// TwinCAT 3 PLC project CraneControl
// ProgramVersion: 3.1.4023.0
// libraries:
//   Tc2_Standard, * (Beckhoff Automation GmbH)
//   Tc2_System, * (Beckhoff Automation GmbH)
//   Tc3_Module, * (Beckhoff Automation GmbH)
//   VisuSymbols,3.5.10.0,System
// project tree:
//   ActuatorLimits/ FB_ActuatorLimits.TcPOU, FB_CartesianVelLimit.TcPOU, G_ActuatorLimits.TcGVL, P_ActuatorLimits.TcPOU, P_CartesianLimit.TcPOU
//   / Class Diagram.TcCD (not stored), GlobalTextList.TcGTLO, PlcTask.TcTTO, Visualization Manager.TcVMO (not stored)
//   ControlBox/ FB_AnalogInputScaling.TcPOU, FB_JoystickInputScaling.TcPOU, G_Buttons.TcGVL, G_ControlBoxInputs.TcGVL, G_Joystick.TcGVL, G_Outputs.TcGVL, G_ScalingParameters.TcGVL (not stored), P_JoystickInput.TcPOU, P_Outputs.TcPOU, ST_AnalogInput.TcDUT (not stored), ST_AnalogInputScaling.TcDUT (not stored), ST_AnalogInputStatus.TcDUT (not stored), ST_JoystickInputScaling.TcDUT (not stored), ST_Parameters.TcDUT
//   HeaveCompensation/ FB_Genr1b.TcPOU, FB_Get3r.TcPOU, G_Heave.TcGVL, P_Heave.TcPOU, P_SetZero.TcPOU
//   KinematicsForwAndInverseMatLab/ eps.TcPOU, eye.TcPOU, FB_ForwardKinematics.TcPOU, FB_InverseKinematics.TcPOU, isequal.TcPOU, MatrixLog3.TcPOU, norm.TcPOU, pinv.TcPOU, pinv_i.TcPOU, svd.TcPOU, svd_e.TcPOU, xaxpy.TcPOU, xaxpy_d.TcPOU, xaxpy_dm.TcPOU, xaxpy_dmy.TcPOU, xaxpy_dmyz.TcPOU, xaxpy_dmyzr.TcPOU, xaxpy_dmyzr5.TcPOU, xdotc.TcPOU, xdotc_i.TcPOU, xnrm2.TcPOU, xnrm2_l.TcPOU, xrot.TcPOU, xrotg.TcPOU, xrot_c.TcPOU, xrot_c5.TcPOU, xscal.TcPOU, xscal_f.TcPOU, xscal_fi.TcPOU, xscal_fiz.TcPOU, xscal_fiz1.TcPOU, rt_floord.TcPOU, rt_ldexp_U1d_U2s32_Yd_s_pw.TcPOU, xdotc_iq.TcPOU, xnrm2_l4.TcPOU, xnrm2_l4b.TcPOU, xscal_fiz1t.TcPOU, xscal_fiz1t4.TcPOU, xswap.TcPOU, xswap_g.TcPOU, xswap_gs.TcPOU
//   JoystickToCartesianVelocity/ FB_JoystickToCartesianVelocity.TcPOU
//   Kinematics_CraneFrame/ FB_ToolpointPositionIntegrator.TcPOU, G_InverseKinematics.TcGVL, G_Toolpoint.TcGVL, P_CartesianVelFromJoystick.TcPOU, P_Kinematics.TcPOU
//   PathGenerator/ FB_PathGenerator.TcPOU, G_Path.TcGVL, P_PathGeneration.TcPOU, P_PathGeneration_1.TcPOU, P_PathGeneration_2.TcPOU, P_PathGeneration_3.TcPOU
//   POUs/ MAIN.TcPOU, P_ModeControl.TcPOU, P_SlaveInputControl.TcPOU, Visualization.TcVIS
//   Sensors/ FB_DistSensorValue2Distance_q4.TcPOU, FB_Encoderval2Angle_q3.TcPOU, G_SensorInput.TcGVL, G_SensorsScaled.TcGVL, P_SensorScaling.TcPOU
//   ServoControl/ FB_PID.TcPOU, FB_PID_Controller.TcPOU, FB_ActuatorVelFeedForward.TcPOU, G_Servo.TcGVL, NormToPulseLenght.TcPOU, ButtonControlPulseLenght.TcPOU, P_CarteseanControllerServoActuation4DOF.TcPOU, P_ManualActuatorTest.TcPOU, P_NormalizeJointVel.TcPOU, P_CartesianController.TcPOU, P_Idle.TcPOU, P_ManualControl.TcPOU, P_VelToPos.TcPOU

CONFIGURATION CraneControl
    RESOURCE PLC ON TwinCAT3
        TASK PlcTask(INTERVAL := T#10ms, PRIORITY := 20);
        PROGRAM MAIN WITH PlcTask : MAIN;
    END_RESOURCE
END_CONFIGURATION

// ---- ControlBox/ST_Parameters.TcDUT
TYPE ST_Parameters :
STRUCT
	fCyclicTime 					: LREAL := 0.01; // [s]
	
	stJoystickInputScalingLeftX 		: ST_JoystickInputScaling := (fMaxInputValue := 20469.0, fMinInputValue := 11924.0, fNeutralInputValue := 16265, fNeutralDeadband := 100.0, fMaxOutputValue := 1.0, fMinOutputValue := -1.0, fNeutralOutputValue := 0.0);
	stJoystickInputScalingLeftY 		: ST_JoystickInputScaling := (fMaxInputValue := 20436.0, fMinInputValue := 11910.0, fNeutralInputValue := 16369, fNeutralDeadband := 100.0, fMaxOutputValue := 1.0, fMinOutputValue := -1.0, fNeutralOutputValue := 0.0);
	stJoystickInputScalingRightX 		: ST_JoystickInputScaling := (fMaxInputValue := 20481.0, fMinInputValue := 11905.0, fNeutralInputValue := 16370, fNeutralDeadband := 100.0, fMaxOutputValue := 1.0, fMinOutputValue := -1.0, fNeutralOutputValue := 0.0);
	stJoystickInputScalingRightY 		: ST_JoystickInputScaling := (fMaxInputValue := 20342.0, fMinInputValue := 12050.0, fNeutralInputValue := 16365, fNeutralDeadband := 100.0, fMaxOutputValue := 1.0, fMinOutputValue := -1.0, fNeutralOutputValue := 0.0);

		
END_STRUCT
END_TYPE

// ---- ActuatorLimits/G_ActuatorLimits.TcGVL
{attribute 'qualified_only'}
VAR_GLOBAL
	fq1Min: LREAL := -1.3;//rad
	fq1Max: LREAL := 1.3;//rad
	fq2Min: LREAL := -1.2;//rad 
	fq2Max: LREAL := 0.65;//rad
	fq3Min: LREAL := 0.15;//rad
	fq3Max: LREAL := 2.5;//rad
	fq4Min: LREAL := 0.0100;//m
	fq4Max: LREAL := 0.1900;//m

	bq1Min: BOOL;  // reached or not
	bq1Max: BOOL;
	bq2Min: BOOL;
	bq2Max: BOOL;
	bq3Min:	BOOL;
	bq3Max: BOOL;
	bq4Min: BOOL;
	bq4Max: BOOL;
	
	// Meassured in crane coordinates with tilt (theta = 0):
	fZMin : LREAL := -0.0500; //m 
	fZMax : LREAL := 0.4000;
	fYMin : LREAL := -0.25;
	fYMax : LREAL := 0.25;
	fXMax : LREAL := 0.45;
	fXMin : LREAL := 0.133;
END_VAR

// ---- ControlBox/G_Buttons.TcGVL
{attribute 'qualified_only'}
VAR_GLOBAL
	bManualModeSelector			AT %I* : BOOL;
	bAutoModeSelector			AT %I* : BOOL;
	//bRedButton					AT %I* : BOOL; Chaned fort extra button on joy stick
	//bGreenButton				AT %I* : BOOL; Chaned fort extra button on joy stick
	bJoystickLeftFrontEnable			AT %I* : BOOL;
	bJoystickRightFrontEnable			AT %I* : BOOL;
	bJoystickLeftEnable			AT %I* : BOOL;
	bJoystickRightEnable		AT %I* : BOOL;
	bSafetyRelayRestartButton   AT %I* : BOOL;
	
	// Analog Inputs
	stJoyLX 					: ST_AnalogInput;
	stJoyLY						: ST_AnalogInput;
	stJoyRX 					: ST_AnalogInput;
	stJoyRY						: ST_AnalogInput;

END_VAR

// ---- ControlBox/G_ControlBoxInputs.TcGVL
{attribute 'qualified_only'}
VAR_GLOBAL
	bManualModeSelector			AT %I* : BOOL;
	bAutoModeSelector			AT %I* : BOOL;
	bRedButton					AT %I* : BOOL;
	bGreenButton				AT %I* : BOOL;
	bJoystickLeftEnable			AT %I* : BOOL;
	bJoystickRightEnable		AT %I* : BOOL;
	bSafetyRelayRestartButton   AT %I* : BOOL;
	
	// Analog Inputs
	stJoyLX 					: ST_AnalogInput;
	stJoyLY						: ST_AnalogInput;
	stJoyRX 					: ST_AnalogInput;
	stJoyRY						: ST_AnalogInput;

END_VAR

// ---- ControlBox/G_Joystick.TcGVL
{attribute 'qualified_only'}
VAR_GLOBAL
	fJoystickLeftNormalizedY 		: LREAL;
	fJoystickLeftNormalizedX 		: LREAL;	
	fJoystickRightNormalizedY 		: LREAL;
	fJoystickRightNormalizedX 		: LREAL;
	
	nJoystickLeftDirectionX 		: DINT;
	nJoystickLeftDirectionY 		: DINT;
	nJoystickRightDirectionX 		: DINT;
	nJoystickRightDirectionY 		: DINT;
	
	bJoystick1InUse : BOOL ;
	bJoystick2InUse : BOOL;
	bJoystick3InUse : BOOL;
	bJoystick4InUse : BOOL;
		
END_VAR

// ---- ControlBox/G_Outputs.TcGVL
{attribute 'qualified_only'}
VAR_GLOBAL
	// PLC Rack
	
	// RIO Rack
	// Digital Outputs
	bGreenButtonLight 			AT %Q* : BOOL;
	bRedButtonLight 			AT %Q* : BOOL;
	// Analog Outputs
	//stWinchValveOutput 		: ST_ValveOutput;
	//stCylValveOutput 			: ST_ValveOutput;
	bSafetyRelayReset		 	AT %Q* : BOOL;
	
END_VAR

// ---- HeaveCompensation/G_Heave.TcGVL
{attribute 'qualified_only'}
VAR_GLOBAL
	fThetaStart : LREAL; //Tipping angle in degrees read at with system at rest
	fTheta : LREAL; //Tipping angle in degrees
	r3x : LREAL; //Vector from tipping point to toolpoint ref in frame coordinate
	r3y : LREAL; //Vector from tipping point to toolpoint ref in frame coordinate
	r3z : LREAL; //Vector from tipping point to toolpoint ref in frame coordinate
	r1bxCrane : LREAL; // Vector from crane base to toolpoint in Crane coordinates
	r1byCrane : LREAL; // Vector from crane base to toolpoint in Crane coordinates
	r1bzCrane : LREAL; // Vector from crane base to toolpoint in Crane coordinates
	bHeaveEnable : BOOL;
	bHeaveActive : BOOL := FALSE;
END_VAR

// ---- Kinematics_CraneFrame/G_InverseKinematics.TcGVL
{attribute 'qualified_only'}
VAR_GLOBAL
	fvXref  : LREAL; // Toolpoint cartesian velocity. From joistick. Used for inv. vel kin and calculate path for pos controller
	fvYref  : LREAL;
	fvZref  : LREAL;
	fq4Dotref : LREAL; //Actuator angular velocity from inverse vel kinematics m/s
	f_q1_ref : LREAL; //Ref angles from inverse position kinematics radians
	f_q2_ref : LREAL;
	f_q3_ref : LREAL;
	bKinematicsSucsessful : BOOL;
END_VAR

// ---- Kinematics_CraneFrame/G_Toolpoint.TcGVL
{attribute 'qualified_only'}
VAR_GLOBAL
	fX  : LREAL; //m
	fY  : LREAL; //m
	fZ  : LREAL; //m
	fXref  : LREAL; // Toolpoint cartesian reference signal position controller
	fYref  : LREAL;//m
	fZref  : LREAL;//m
END_VAR

// ---- PathGenerator/G_Path.TcGVL
{attribute 'qualified_only'}
VAR_GLOBAL
	bPathRunning  : BOOL;
	bPathFinnish : BOOL;
	bStartPath : BOOL;
	tTime : LREAL;
	bPathActivated : BOOL; // HMI path or Joistick
END_VAR

// ---- Sensors/G_SensorInput.TcGVL
{attribute 'qualified_only'}
VAR_GLOBAL
	fEncoder1Rad AT %I* : REAL;
	fEncoder2Rad AT %I* : REAL;
	fEncoder3Rad AT %I* : REAL;
	fTelescopeDistance_mm AT %I* : REAL;
	fXRotDeg AT %I* : REAL;
	fYRotDeg AT %I* : REAL;
	bSensorDataLost : BOOL;
END_VAR

// ---- Sensors/G_SensorsScaled.TcGVL
{attribute 'qualified_only'}
VAR_GLOBAL
	q1: REAL;
	q2  : REAL;
	q3  : REAL;
	q4 : REAL;
	q1Dot: REAL;
	q2Dot  : REAL;
	q3Dot  : REAL;
	q4Dot : REAL;
END_VAR

// ---- ServoControl/G_Servo.TcGVL
{attribute 'qualified_only'}
VAR_GLOBAL
	nServoPulseLenght1		AT %Q* : UINT;
	nServoPulseLenght2		AT %Q* : UINT;
	nServoPulseLenght3		AT %Q* : UINT;
	nServoPulseLenght4		AT %Q* : UINT;
	nServoPulseLenght5		AT %Q* : UINT;
	nServoPulseLenght6		AT %Q* : UINT;
	
	fNormalizedActuatorVelFeedForward_q1Dot : LREAL;
	fNormalizedActuatorVelFeedForward_q2Dot : LREAL;
	fNormalizedActuatorVelFeedForward_q3Dot : LREAL;
	fNormalizedActuatorVelFeedForward_q4Dot : LREAL;
	
	q1_position_error_part : LREAL;
	q2_position_error_part : LREAL;
	q3_position_error_part : LREAL;
	q4_position_error_part : LREAL;
	
	f_u_q1 :LREAL;
	f_u_q2 :LREAL;
	f_u_q3 :LREAL;
	f_u_q4 :LREAL; 
	
	
	//Temp for servo test:
	bStartSinus : BOOL;
	bSinusActive : BOOL;
	
END_VAR

// ---- POUs/MAIN.TcPOU
PROGRAM MAIN
VAR
END_VAR

P_ModeControl();

END_PROGRAM

// ---- POUs/P_ModeControl.TcPOU
PROGRAM P_ModeControl
VAR
	bAllowSinusInManualMode : BOOL;
END_VAR


// ONLY SET TRUE FOR ACTUATOR TEST IN MANUAL MODE:
bAllowSinusInManualMode := FALSE;



P_SensorScaling(); // Scaling sensor signals to mach q1,q2,q3,q4
P_Kinematics(); // Toolpoint position based on joint angles
P_JoystickInput(); // Normalize joistick signals from raw to -1 to 1


IF G_Buttons.bManualModeSelector AND NOT(G_Buttons.bAutoModeSelector) THEN // Manual mode
	
	//Only for actuationg the joints with open loop sinus
	IF G_Servo.bSinusActive AND bAllowSinusInManualMode THEN
		P_ManualActuatorTest();
	ELSE
		P_ManualControl();
	END_IF
	
	
	
	P_ActuatorLimits(); // Checking sensors and light lamps in HMI, preventing crashes is ONLY in auto mode
ELSIF NOT(G_Buttons.bManualModeSelector) AND G_Buttons.bAutoModeSelector AND NOT(G_SensorInput.bSensorDataLost) THEN // Auto Mode
	// Choose joystick OR PathGeneration

	IF G_Path.bPathActivated THEN
		//P_PathGeneration_1();  // 4 DOF
		P_PathGeneration_2();  // 4 DOF (3 dof test different telescope)
		//P_PathGeneration();  // 3 DOF
	ELSE
		P_CartesianVelFromJoystick();		
	END_IF

	
	P_CartesianLimit(); // Stops velocity ref if outside boundaries


	IF G_Heave.bHeaveEnable THEN
		P_Heave();
		G_Heave.bHeaveActive := TRUE;
	ELSE
		G_Heave.bHeaveActive := FALSE;
		P_VelToPos(); //Integrates pos to vel if 
	END_IF
	
	P_CartesianController();
ELSE // ModeButton in zero position
	P_Idle();
	P_SetZero();
	G_Heave.bHeaveActive := FALSE;
END_IF


P_Outputs(); //Lights on control box

END_PROGRAM

// ---- Sensors/P_SensorScaling.TcPOU
PROGRAM P_SensorScaling
VAR
		fbEncoderval2Angleq3 : FB_Encoderval2Angle_q3;
		fbDistSensorValue2Distance_q4 : FB_DistSensorValue2Distance_q4;

	
	// Temp variables for checking sensor comunication
	tempTOF1: LREAL;
	tempTOF11: LREAL;
	tempCounter: DINT := 0;

END_VAR

fbEncoderval2Angleq3(theta_i := G_SensorInput.fEncoder3Rad ,
					q3 => G_SensorsScaled.q3);
					
					
G_SensorsScaled.q1 := -G_SensorInput.fEncoder1Rad;
G_SensorsScaled.q2 := -G_SensorInput.fEncoder2Rad;



fbDistSensorValue2Distance_q4(fSensorValue := G_SensorInput.fTelescopeDistance_mm,
							f_q4 => G_SensorsScaled.q4);								
// TEMP FOR 3 DOF
//G_SensorsScaled.q4 := 0;
			

/////////////////////////////////////////////////////////////////////////////
// Check if sensors are comunicating and lighting RED LED communication lost	
tempTOF1 := G_SensorInput.fTelescopeDistance_mm;
IF tempTOF1 = tempTOF11 THEN
	tempCounter := tempCounter +1;
ELSE
	tempCounter := 0;
END_IF
tempTOF11 := G_SensorInput.fTelescopeDistance_mm;

IF tempCounter > 50 THEN
	G_SensorInput.bSensorDataLost := TRUE;
ELSE
	G_SensorInput.bSensorDataLost := FALSE;
END_IF
//////////////////////////////////////////////////////////////////////////////

END_PROGRAM

// ---- Sensors/FB_Encoderval2Angle_q3.TcPOU
FUNCTION_BLOCK FB_Encoderval2Angle_q3
VAR_INPUT
	theta_i: REAL;
END_VAR
VAR_OUTPUT
	q3: REAL;
END_VAR
VAR_TEMP
	ll: REAL;
	a: REAL;
	q3_tmp: REAL;
	temp1: REAL;
	temp2: REAL;
END_VAR

(* MATLAB Function: '<Root>/MATLAB Function' *)
(* Validated with physical measurements on crane from 0 - 180 deg *)
(* MATLAB Function 'MATLAB Function': '<S1>:1' *)
(* Constant Leght all mm: *)
(* '<S1>:1:6' theta_i_init = 2.3527; *)
(* start angle when piston is fully extracted *)
(* '<S1>:1:7' theta_k_init = 3.9706; *)
(* start angle when piston is fully extracted *)
(* '<S1>:1:8' Theta_I = theta_i_init + theta_i; *)
(* '<S1>:1:10' lh = 116.62; *)
(* '<S1>:1:11' li = 121.93; *)
(* '<S1>:1:12' lj = 13.34; *)
(* '<S1>:1:13' lk = 30; *)
(* '<S1>:1:14' lm = 20; *)
(* '<S1>:1:15' ln = 16; *)
(* '<S1>:1:16' theta_h = real(acos((lh^2+lj^2-li^2)/(2*lh*lj))); *)
(* Based on input: *)
(* Cylinder lenght: *)
(* '<S1>:1:20' xk = sqrt(lh^2+lk^2-2*lh*lk*cos(Theta_I)); *)

// PHMH ADDED BECAUSE BUNCTION DOES NOT HANDLE POSITIVE VALUES. Posistive values not possible after caluibration
IF theta_i >= 0 THEN
	theta_i := -0.00001;
ELSIF theta_i <= -1.5 THEN
	theta_i := -1.5;
END_IF




temp1 := COS(theta_i + 2.3527);
IF ABS(temp1) > 1 THEN
	temp1 := 1;
END_IF



a := SQRT(14500.224400000001 - (temp1 * 6997.2000000000007));
(* '<S1>:1:22' theta_j = theta_h-Theta_I; *)
(* '<S1>:1:23' ll = sqrt(lj^2+lk^2-2*lj*lk*cos(theta_j)); *)
temp2 := COS(1.9282807448254589 - (theta_i + 2.3527));
ll := SQRT(1077.9556 - (temp2 * 800.4));
(* '<S1>:1:25' theta_n = real(acos((ll^2+ln^2-lm^2)/(2*ll*ln))); *)
(* '<S1>:1:26' theta_l = acos((li^2+ll^2-xk^2)/(2*li*ll)); *)
(* '<S1>:1:27' theta_k = theta_n + theta_l; *)
(* '<S1>:1:28' q3 = theta_k-theta_k_init; *)
(* - init so output start at 0 *)
q3_tmp := ll * ll;
(* Outport: '<Root>/q3' incorporates:
 *  MATLAB Function: '<Root>/MATLAB Function' *)
q3 := -((ACOS(((q3_tmp + 256.0) - 400.0) / ((2.0 * ll) * 16.0)) + ACOS(((q3_tmp + 14866.924900000002) - (a * a)) / (243.86 * ll))) - 3.9706);

END_FUNCTION_BLOCK

// ---- Sensors/FB_DistSensorValue2Distance_q4.TcPOU
FUNCTION_BLOCK FB_DistSensorValue2Distance_q4
VAR_INPUT
	fSensorValue : REAL;
END_VAR
VAR_OUTPUT
	f_q4 : REAL;
END_VAR
VAR
DistSensorVal : REAL := 190; //mm
//Meassured value (Can be ecalibrated by looking in G_SensorInput and reading min and max telescope dist):
DistSensorMin : REAL  := 8.5; //mm
DistSensorMax : REAL := 193; //mm
 
q4Min : REAL := 167.25; //Maching with physical measurement 
q4Max : REAL := 367.25;//200 mm work space
END_VAR

f_q4 :=  ((fSensorValue-DistSensorMin)/(DistSensorMax-DistSensorMin)*(q4Max-q4Min))/1000;//m

END_FUNCTION_BLOCK

// ---- Kinematics_CraneFrame/P_Kinematics.TcPOU
PROGRAM P_Kinematics
VAR
fbForwardKinematics	: FB_ForwardKinematics;
END_VAR

fbForwardKinematics(q1 := G_SensorsScaled.q1, 
					q2 := G_SensorsScaled.q2,
					q3 := G_SensorsScaled.q3,
					q4 := G_SensorsScaled.q4,
					x => G_Toolpoint.fX,
					y => G_Toolpoint.fY,
					z => G_Toolpoint.fZ);

END_PROGRAM

// ---- KinematicsForwAndInverseMatLab/FB_ForwardKinematics.TcPOU
FUNCTION_BLOCK FB_ForwardKinematics
VAR_INPUT
    q1: LREAL;
    q2: LREAL;
    q3: LREAL;
    q4: LREAL;
END_VAR
VAR_OUTPUT
    x: LREAL;
    y: LREAL;
    z: LREAL;
END_VAR
VAR
    b: ARRAY [0..15] OF LREAL := [1.0,0.0,0.0,0.0,0.0,1.0,0.0,0.0,0.0,0.0,1.0,0.0,0.31920000000000004,0.02686,
        0.15515,1.0];
    c: ARRAY [0..35] OF LREAL := [0.0,0.0,1.0,0.0,0.0,0.0,0.0,1.0,0.0,-0.1569,0.0,-0.02745,0.0,1.0,0.0,-0.1569,0.0,
        0.15195,0.0,0.0,0.0,1.0,0.0,0.0,0.0,1.0,0.0,-0.15515,0.0,0.31920000000000004,0.0,0.0,1.0,0.02686,
        -0.31920000000000004,0.0];
    e_a: ARRAY [0..8] OF SINT := [1,0,0,0,1,0,0,0,1];
END_VAR
VAR_TEMP
    thetalist: ARRAY [0..5] OF LREAL;
    T: ARRAY [0..15] OF LREAL;
    i: DINT;
    se3mat: ARRAY [0..15] OF LREAL;
    omgmat: ARRAY [0..8] OF LREAL;
    a: ARRAY [0..15] OF LREAL;
    c_a: LREAL;
    V: ARRAY [0..5] OF LREAL;
    b_R: ARRAY [0..8] OF LREAL;
    b_omgmat: ARRAY [0..8] OF LREAL;
    d_a: LREAL;
    b_I: ARRAY [0..8] OF SINT;
    omgtheta_tmp: ARRAY [0..2] OF LREAL;
    thetalist_0: LREAL;
    a_0: ARRAY [0..15] OF LREAL;
    i_0: DINT;
    a_tmp_tmp: DINT;
    omgmat_tmp: DINT;
    R_tmp: DINT;
    c_a_tmp: LREAL;
    b_a_tmp: LREAL;
END_VAR

(* Lenght from assy drawing *)
(* MATLAB Function 'MATLAB Function': '<S1>:1' *)
(* '<S1>:1:4' l1 = 156.9/1000; *)
(* '<S1>:1:5' l2 = 27.45/1000; *)
(* '<S1>:1:6' l3 = 179.4/1000; *)
(* '<S1>:1:7' l4 = 26.86/1000; *)
(* From Telescope drawing (IN assy drawing) *)
(* l5 = 163.43;  *)
(* '<S1>:1:10' l5 = 167.25/1000; *)
(* Corrected after sensor calibration  *)
(* '<S1>:1:11' l6 = 1.75/1000; *)
(* mm *)
(* '<S1>:1:12' W1 = -l2+l3+l5; *)
(* '<S1>:1:13' W2 = l4; *)
(* '<S1>:1:14' W3 = l1-l6; *)
(* Position of each joint *)
(* '<S1>:1:18' a1 = [0; 0; 0]; *)
(* '<S1>:1:19' a2 = [-l2; 0; l1]; *)
(* '<S1>:1:20' a3 = [-l2+l3; 0; l1]; *)
(* '<S1>:1:21' a4 = [W1; W2; W3]; *)
(* '<S1>:1:22' a5 = [W1; W2; W3]; *)
(* '<S1>:1:23' a6 = [W1; W2; W3]; *)
(* Screw axis of ech joint *)
(* '<S1>:1:26' Sw1 = [0; 0; 1]; *)
(* '<S1>:1:27' Sw2 = [0; 1; 0]; *)
(* '<S1>:1:28' Sw3 = [0; 1; 0]; *)
(* '<S1>:1:29' Sw4 = [0; 0; 0]; *)
(* '<S1>:1:30' Sw5 = [0; 1; 0]; *)
(* '<S1>:1:31' Sw6 = [0; 0; 1]; *)
(* '<S1>:1:33' Sv1 = cross(a1,Sw1); *)
(* '<S1>:1:34' Sv2 = cross(a2,Sw2); *)
(* '<S1>:1:35' Sv3 = cross(a3,Sw3); *)
(* '<S1>:1:36' Sv4 = [1;0;0]; *)
(* translation along xaxis *)
(* '<S1>:1:37' Sv5 = cross(a5,Sw5); *)
(* '<S1>:1:38' Sv6 = cross(a6,Sw6); *)
(* '<S1>:1:40' S1 = [Sw1;Sv1]; *)
(* '<S1>:1:41' S2 = [Sw2;Sv2]; *)
(* '<S1>:1:42' S3 = [Sw3;Sv3]; *)
(* '<S1>:1:43' S4 = [Sw4;Sv4]; *)
(* '<S1>:1:44' S5 = [Sw5;Sv5]; *)
(* '<S1>:1:45' S6 = [Sw6;Sv6]; *)
(* '<S1>:1:47' M = [[1 0 0 W1]; *)
(* '<S1>:1:48'     [0 1 0 W2]; *)
(* '<S1>:1:49'     [0 0 1 W3]; *)
(* '<S1>:1:50'     [0 0 0 1];]; *)
(* MATLAB Function: '<Root>/MATLAB Function' *)
FOR i_0 := 0 TO 15 DO 
    T[i_0] := b[i_0];
END_FOR;
(* Joints:  *)
(* '<S1>:1:55' q5 = 0; *)
(* '<S1>:1:56' q6 = 0; *)
(* '<S1>:1:58' thetalist = [q1; q2 ; q3; q4; q5; q6]; *)
thetalist[0] := q1;
thetalist[1] := q2;
thetalist[2] := q3;
thetalist[3] := q4;
thetalist[4] := 0.0;
thetalist[5] := 0.0;
(* '<S1>:1:59' Slist = [S1,S2,S3,S4,S5,S6]; *)
(* '<S1>:1:63' T = M; *)
(* '<S1>:1:65' for i = 6: -1: 1 *)
(* MATLAB Function: '<Root>/MATLAB Function' *)
se3mat[0] := 0.0;
se3mat[5] := 0.0;
se3mat[10] := 0.0;
se3mat[3] := 0.0;
se3mat[7] := 0.0;
se3mat[11] := 0.0;
se3mat[15] := 0.0;
(* MATLAB Function: '<Root>/MATLAB Function' *)
(* MATLAB Function: '<Root>/MATLAB Function' *)
FOR i := 0 TO 5 DO 
    (* 6 = number of joints *)
    (* '<S1>:1:67' T = MatrixExp6(VecTose3(Slist(:, i) * thetalist(i))) * T; *)
    thetalist_0 := thetalist[5 - i];
    FOR i_0 := 0 TO 5 DO 
        V[i_0] := c[((5 - i) * 6) + i_0] * thetalist_0;
    END_FOR;
    (* *** CHAPTER 3: RIGID-BODY MOTIONS *** *)
    (* Takes a 6-vector (representing a spatial velocity). *)
    (* Returns the corresponding 4x4 se(3) matrix. *)
    (* Example Input: *)
    
    (* clear; clc; *)
    (* V = [1; 2; 3; 4; 5; 6]; *)
    (* se3mat = VecTose3(V) *)
    
    (* Output: *)
    (* se3mat = *)
    (* 0    -3     2     4 *)
    (* 3     0    -1     5 *)
    (* -2     1     0     6 *)
    (* 0     0     0     0  *)
    (* 'VecTose3:18' se3mat = [VecToso3(V(1: 3)), V(4: 6); 0, 0, 0, 0]; *)
    (* *** CHAPTER 3: RIGID-BODY MOTIONS *** *)
    (* Takes a 3-vector (angular velocity). *)
    (* Returns the skew symmetric matrix in so(3). *)
    (* Example Input: *)
    
    (* clear; clc; *)
    (* omg = [1; 2; 3]; *)
    (* so3mat = VecToso3(omg) *)
    
    (* Output: *)
    (* so3mat = *)
    (* 0    -3     2 *)
    (* 3     0    -1 *)
    (* -2     1     0 *)
    (* 'VecToso3:17' so3mat = [0, -omg(3), omg(2); omg(3), 0, -omg(1); -omg(2), omg(1), 0]; *)
    se3mat[4] :=  -V[2];
    se3mat[8] := V[1];
    se3mat[1] := V[2];
    se3mat[9] :=  -V[0];
    se3mat[2] :=  -V[1];
    se3mat[6] := V[0];
    se3mat[12] := V[3];
    se3mat[13] := V[4];
    se3mat[14] := V[5];
    (* *** CHAPTER 3: RIGID-BODY MOTIONS *** *)
    (* Takes a se(3) representation of exponential coordinates. *)
    (* Returns a T matrix in SE(3) that is achieved by traveling along/about the  *)
    (* screw axis S for a distance theta from an initial configuration T = I. *)
    (* Example Input: *)
    
    (* clear; clc; *)
    (* se3mat = [ 0,      0,       0,      0; *)
    (* 0,      0, -1.5708, 2.3562; *)
    (* 0, 1.5708,       0, 2.3562; *)
    (* 0,      0,       0,      0] *)
    (* T = MatrixExp6(se3mat) *)
    
    (* Output: *)
    (* T = *)
    (* 1.0000         0         0         0 *)
    (* 0    0.0000   -1.0000   -0.0000 *)
    (* 0    1.0000    0.0000    3.0000 *)
    (* 0         0         0    1.0000  *)
    (* 'MatrixExp6:22' omgtheta = so3ToVec(se3mat(1: 3, 1: 3)); *)
    (* *** CHAPTER 3: RIGID-BODY MOTIONS *** *)
    (* Takes a 3x3 skew-symmetric matrix (an element of so(3)). *)
    (* Returns the corresponding 3-vector (angular velocity). *)
    (* Example Input:  *)
    
    (* clear; clc; *)
    (* so3mat = [[0, -3, 2]; [3, 0, -1]; [-2, 1, 0]]; *)
    (* omg = so3ToVec(so3mat)   *)
    
    (* Output: *)
    (* omg = *)
    (* 1 *)
    (* 2 *)
    (* 3 *)
    (* 'so3ToVec:17' omg = [so3mat(3, 2); so3mat(1, 3); so3mat(2, 1)]; *)
    omgtheta_tmp[0] := V[0];
    omgtheta_tmp[1] := V[1];
    omgtheta_tmp[2] := V[2];
    (* 'MatrixExp6:23' if NearZero(norm(omgtheta)) *)
    (* *** BASIC HELPER FUNCTIONS *** *)
    (* Takes a scalar. *)
    (* Checks if the scalar is small enough to be neglected. *)
    (* Example Input: *)
    
    (* clear; clc; *)
    (* near = -1e-7; *)
    (* judge = NearZero(near) *)
    
    (* Output: *)
    (* judge = *)
    (* 1 *)
    (* 'NearZero:15' judge = norm(near) < 1e-6; *)
    thetalist_0 := norm(x := omgtheta_tmp);
    d_a := ABS(thetalist_0);
    IF d_a < 1.0E-6 THEN 
        (* 'MatrixExp6:24' T = [eye(3), se3mat(1: 3, 4); 0, 0, 0, 1]; *)
        FOR i_0 := 0 TO 8 DO 
            b_I[i_0] := 0;
        END_FOR;
        b_I[0] := 1;
        b_I[4] := 1;
        b_I[8] := 1;
        FOR i_0 := 0 TO 2 DO 
            R_tmp := DWORD_TO_DINT(SHL(DINT_TO_DWORD(i_0), 2));
            a[R_tmp] := SINT_TO_LREAL(b_I[3 * i_0]);
            a[R_tmp + 1] := SINT_TO_LREAL(b_I[(3 * i_0) + 1]);
            a[R_tmp + 2] := SINT_TO_LREAL(b_I[(3 * i_0) + 2]);
            a[i_0 + 12] := se3mat[i_0 + 12];
        END_FOR;
        a[3] := 0.0;
        a[7] := 0.0;
        a[11] := 0.0;
        a[15] := 1.0;
    ELSE 
        (* 'MatrixExp6:25' else *)
        (* 'MatrixExp6:26' [omghat, theta] = AxisAng3(omgtheta); *)
        (* *** CHAPTER 3: RIGID-BODY MOTIONS *** *)
        (* Takes A 3-vector of exponential coordinates for rotation. *)
        (* Returns the unit rotation axis omghat and the corresponding rotation  *)
        (* angle theta. *)
        (* Example Input: *)
        
        (* clear; clc; *)
        (* expc3 = [1; 2; 3]; *)
        (* [omghat, theta] = AxisAng3(expc3)   *)
        
        (* Output: *)
        (* omghat = *)
        (* 0.2673 *)
        (* 0.5345 *)
        (* 0.8018 *)
        (* theta = *)
        (* 3.7417 *)
        (* 'AxisAng3:20' theta = norm(expc3); *)
        (* 'AxisAng3:21' omghat = expc3 / theta; *)
        (* 'MatrixExp6:27' omgmat = se3mat(1: 3, 1: 3) / theta; *)
        FOR i_0 := 0 TO 2 DO 
            omgmat_tmp := DWORD_TO_DINT(SHL(DINT_TO_DWORD(i_0), 2));
            omgmat[3 * i_0] := se3mat[omgmat_tmp] / thetalist_0;
            omgmat[(3 * i_0) + 1] := se3mat[omgmat_tmp + 1] / thetalist_0;
            omgmat[(3 * i_0) + 2] := se3mat[omgmat_tmp + 2] / thetalist_0;
        END_FOR;
        (* 'MatrixExp6:28' T = [MatrixExp3(se3mat(1: 3, 1: 3)), ... *)
        (* 'MatrixExp6:29'          (eye(3) * theta + (1 - cos(theta)) * omgmat ... *)
        (* 'MatrixExp6:30'           + (theta - sin(theta)) * omgmat * omgmat) ... *)
        (* 'MatrixExp6:31'             * se3mat(1: 3, 4) / theta; *)
        (* 'MatrixExp6:32'          0, 0, 0, 1]; *)
        b_a_tmp := COS(thetalist_0);
        c_a_tmp := SIN(thetalist_0);
        c_a := thetalist_0 - c_a_tmp;
        (* *** CHAPTER 3: RIGID-BODY MOTIONS *** *)
        (* Takes a 3x3 so(3) representation of exponential coordinates. *)
        (* Returns R in SO(3) that is achieved by rotating about omghat by theta  *)
        (* from an initial orientation R = I. *)
        (* Example Input: *)
        
        (* clear; clc; *)
        (* so3mat = [[0, -3, 2]; [3, 0, -1]; [-2, 1, 0]]; *)
        (* R = MatrixExp3(so3mat)   *)
        
        (* Output: *)
        (* R = *)
        (* -0.6949    0.7135    0.0893 *)
        (* -0.1920   -0.3038    0.9332 *)
        (* 0.6930    0.6313    0.3481 *)
        (* 'MatrixExp3:18' omgtheta = so3ToVec(so3mat); *)
        (* *** CHAPTER 3: RIGID-BODY MOTIONS *** *)
        (* Takes a 3x3 skew-symmetric matrix (an element of so(3)). *)
        (* Returns the corresponding 3-vector (angular velocity). *)
        (* Example Input:  *)
        
        (* clear; clc; *)
        (* so3mat = [[0, -3, 2]; [3, 0, -1]; [-2, 1, 0]]; *)
        (* omg = so3ToVec(so3mat)   *)
        
        (* Output: *)
        (* omg = *)
        (* 1 *)
        (* 2 *)
        (* 3 *)
        (* 'so3ToVec:17' omg = [so3mat(3, 2); so3mat(1, 3); so3mat(2, 1)]; *)
        (* 'MatrixExp3:19' if NearZero(norm(omgtheta)) *)
        (* *** BASIC HELPER FUNCTIONS *** *)
        (* Takes a scalar. *)
        (* Checks if the scalar is small enough to be neglected. *)
        (* Example Input: *)
        
        (* clear; clc; *)
        (* near = -1e-7; *)
        (* judge = NearZero(near) *)
        
        (* Output: *)
        (* judge = *)
        (* 1 *)
        (* 'NearZero:15' judge = norm(near) < 1e-6; *)
        IF d_a < 1.0E-6 THEN 
            (* 'MatrixExp3:20' R = eye(3); *)
            FOR i_0 := 0 TO 8 DO 
                b_R[i_0] := 0.0;
            END_FOR;
            b_R[0] := 1.0;
            b_R[4] := 1.0;
            b_R[8] := 1.0;
        ELSE 
            (* 'MatrixExp3:21' else *)
            (* 'MatrixExp3:22' [omghat, theta] = AxisAng3(omgtheta); *)
            (* *** CHAPTER 3: RIGID-BODY MOTIONS *** *)
            (* Takes A 3-vector of exponential coordinates for rotation. *)
            (* Returns the unit rotation axis omghat and the corresponding rotation  *)
            (* angle theta. *)
            (* Example Input: *)
            
            (* clear; clc; *)
            (* expc3 = [1; 2; 3]; *)
            (* [omghat, theta] = AxisAng3(expc3)   *)
            
            (* Output: *)
            (* omghat = *)
            (* 0.2673 *)
            (* 0.5345 *)
            (* 0.8018 *)
            (* theta = *)
            (* 3.7417 *)
            (* 'AxisAng3:20' theta = norm(expc3); *)
            (* 'AxisAng3:21' omghat = expc3 / theta; *)
            (* 'MatrixExp3:23' omgmat = so3mat / theta; *)
            FOR i_0 := 0 TO 2 DO 
                omgmat_tmp := DWORD_TO_DINT(SHL(DINT_TO_DWORD(i_0), 2));
                b_omgmat[3 * i_0] := se3mat[omgmat_tmp] / thetalist_0;
                b_omgmat[(3 * i_0) + 1] := se3mat[omgmat_tmp + 1] / thetalist_0;
                b_omgmat[(3 * i_0) + 2] := se3mat[omgmat_tmp + 2] / thetalist_0;
            END_FOR;
            (* 'MatrixExp3:24' R = eye(3) + sin(theta) * omgmat + (1 - cos(theta)) * omgmat * omgmat; *)
            FOR i_0 := 0 TO 8 DO 
                b_I[i_0] := 0;
            END_FOR;
            b_I[0] := 1;
            b_I[4] := 1;
            b_I[8] := 1;
            FOR i_0 := 0 TO 2 DO 
                FOR omgmat_tmp := 0 TO 2 DO 
                    R_tmp := (3 * omgmat_tmp) + i_0;
                    b_R[R_tmp] := (((((1.0 - b_a_tmp) * b_omgmat[i_0 + 3]) * b_omgmat[(3 * omgmat_tmp) + 1]) + (((1.0 - b_a_tmp) * b_omgmat[i_0]) * b_omgmat[3 * omgmat_tmp])) + ((b_omgmat[i_0 + 6] * (1.0 - b_a_tmp)) * b_omgmat[(3 * omgmat_tmp) + 2])) + ((b_omgmat[R_tmp] * c_a_tmp) + SINT_TO_LREAL(b_I[R_tmp]));
                END_FOR;
            END_FOR;
        END_IF;
        FOR i_0 := 0 TO 2 DO 
            d_a := 0.0;
            FOR omgmat_tmp := 0 TO 2 DO 
                R_tmp := (3 * omgmat_tmp) + i_0;
                d_a := ((((((omgmat[i_0 + 3] * c_a) * omgmat[(3 * omgmat_tmp) + 1]) + ((c_a * omgmat[i_0]) * omgmat[3 * omgmat_tmp])) + ((omgmat[i_0 + 6] * c_a) * omgmat[(3 * omgmat_tmp) + 2])) + ((SINT_TO_LREAL(e_a[R_tmp]) * thetalist_0) + (omgmat[R_tmp] * (1.0 - b_a_tmp)))) * se3mat[omgmat_tmp + 12]) + d_a;
                a[omgmat_tmp + (i_0 * 4)] := b_R[(3 * i_0) + omgmat_tmp];
            END_FOR;
            a[i_0 + 12] := d_a / thetalist_0;
        END_FOR;
        a[3] := 0.0;
        a[7] := 0.0;
        a[11] := 0.0;
        a[15] := 1.0;
    END_IF;
    FOR i_0 := 0 TO 3 DO 
        FOR omgmat_tmp := 0 TO 3 DO 
            a_tmp_tmp := DWORD_TO_DINT(SHL(DINT_TO_DWORD(omgmat_tmp), 2));
            R_tmp := i_0 + a_tmp_tmp;
            a_0[R_tmp] := 0.0;
            a_0[R_tmp] := a_0[R_tmp] + (T[a_tmp_tmp] * a[i_0]);
            a_0[R_tmp] := (T[a_tmp_tmp + 1] * a[i_0 + 4]) + a_0[R_tmp];
            a_0[R_tmp] := (T[a_tmp_tmp + 2] * a[i_0 + 8]) + a_0[R_tmp];
            a_0[R_tmp] := (T[a_tmp_tmp + 3] * a[i_0 + 12]) + a_0[R_tmp];
        END_FOR;
    END_FOR;
    FOR i_0 := 0 TO 15 DO 
        T[i_0] := a_0[i_0];
    END_FOR;
END_FOR;
(* Outport: '<Root>/x' incorporates:
 *  MATLAB Function: '<Root>/MATLAB Function' *)
(* '<S1>:1:69' x = T(1,4); *)
(* '<S1>:1:70' y = T(2,4); *)
(* '<S1>:1:71' z = T(3,4); *)
x := T[12];
(* Outport: '<Root>/y' incorporates:
 *  MATLAB Function: '<Root>/MATLAB Function' *)
y := T[13];
(* Outport: '<Root>/z' incorporates:
 *  MATLAB Function: '<Root>/MATLAB Function' *)
z := T[14];

END_FUNCTION_BLOCK

// ---- KinematicsForwAndInverseMatLab/norm.TcPOU
FUNCTION norm : LREAL
VAR_INPUT
    x: ARRAY [0..2] OF LREAL;
END_VAR
VAR
    scale: LREAL;
    absxk: LREAL;
    t: LREAL;
END_VAR

scale := 3.3121686421112381E-170;
absxk := ABS(x[0]);
IF absxk > 3.3121686421112381E-170 THEN 
    norm := 1.0;
    scale := absxk;
ELSE 
    t := absxk / 3.3121686421112381E-170;
    norm := t * t;
END_IF;
absxk := ABS(x[1]);
IF absxk > scale THEN 
    t := scale / absxk;
    norm := ((norm * t) * t) + 1.0;
    scale := absxk;
ELSE 
    t := absxk / scale;
    norm := (t * t) + norm;
END_IF;
absxk := ABS(x[2]);
IF absxk > scale THEN 
    t := scale / absxk;
    norm := ((norm * t) * t) + 1.0;
    scale := absxk;
ELSE 
    t := absxk / scale;
    norm := (t * t) + norm;
END_IF;
norm := scale * SQRT(norm);

END_FUNCTION

// ---- ControlBox/P_JoystickInput.TcPOU
PROGRAM P_JoystickInput
VAR
	fbJoystickLeftVert 					: FB_JoystickInputScaling;
	fbJoystickLeftHor 					: FB_JoystickInputScaling;
	
	fbJoystickRightVert 				: FB_JoystickInputScaling;
	fbJoystickRightHor 					: FB_JoystickInputScaling;
	
	bEnableJoystick : BOOL;
		
END_VAR

bEnableJoystick := G_Buttons.bManualModeSelector OR G_Buttons.bAutoModeSelector;

fbJoystickLeftVert(
	bEnable := bEnableJoystick,
	nRawInput := G_Buttons.stJoyLY.nValue,
	stJoystickInputScaling := G_ScalingParameters.stParam.stJoystickInputScalingLeftY,
	fNormalizedOutput => G_Joystick.fJoystickLeftNormalizedY
);

IF G_Joystick.fJoystickLeftNormalizedY < 0 THEN
	G_Joystick.nJoystickLeftDirectionY := -1;
ELSIF G_Joystick.fJoystickLeftNormalizedY > 0 THEN
	G_Joystick.nJoystickLeftDirectionY := 1;	
END_IF

fbJoystickLeftHor(
	bEnable := bEnableJoystick,
	nRawInput := G_Buttons.stJoyLX.nValue,
	stJoystickInputScaling := G_ScalingParameters.stParam.stJoystickInputScalingLeftX,
	fNormalizedOutput => G_Joystick.fJoystickLeftNormalizedX
);

IF G_Joystick.fJoystickLeftNormalizedX < 0 THEN
	G_Joystick.nJoystickLeftDirectionX := 1;
ELSIF G_Joystick.fJoystickLeftNormalizedX > 0 THEN
	G_Joystick.nJoystickLeftDirectionX := -1;	
END_IF


fbJoystickRightVert(
	bEnable := bEnableJoystick,
	nRawInput := G_Buttons.stJoyRY.nValue,
	stJoystickInputScaling := G_ScalingParameters.stParam.stJoystickInputScalingRightY,
	fNormalizedOutput => G_Joystick.fJoystickRightNormalizedY
);

IF G_Joystick.fJoystickRightNormalizedY > 0 THEN
	G_Joystick.nJoystickRightDirectionY := -1;
ELSIF G_Joystick.fJoystickRightNormalizedY < 0 THEN
	G_Joystick.nJoystickRightDirectionY := 1;	
END_IF



fbJoystickRightHor(
	bEnable := bEnableJoystick,
	nRawInput := G_Buttons.stJoyRX.nValue,
	stJoystickInputScaling := G_ScalingParameters.stParam.stJoystickInputScalingRightX,
	fNormalizedOutput => G_Joystick.fJoystickRightNormalizedX
);

IF G_Joystick.fJoystickRightNormalizedX < 0 THEN
	G_Joystick.nJoystickRightDirectionX := 1;
ELSIF G_Joystick.fJoystickRightNormalizedX > 0 THEN
	G_Joystick.nJoystickRightDirectionX := -1;	
END_IF


// Activate bool for each joystick
IF G_Joystick.fJoystickRightNormalizedX < 0 OR G_Joystick.fJoystickRightNormalizedX > 0 THEN
	G_Joystick.bJoystick1InUse := TRUE;
ELSE
	G_Joystick.bJoystick1InUse := FALSE;
END_IF

IF G_Joystick.fJoystickRightNormalizedY < 0 OR G_Joystick.fJoystickRightNormalizedY > 0 THEN
	G_Joystick.bJoystick2InUse := TRUE;
ELSE
	G_Joystick.bJoystick2InUse := FALSE;
END_IF

IF G_Joystick.fJoystickLeftNormalizedX < 0 OR G_Joystick.fJoystickLeftNormalizedX > 0 THEN
	G_Joystick.bJoystick3InUse := TRUE;
ELSE
	G_Joystick.bJoystick3InUse := FALSE;
END_IF

IF G_Joystick.fJoystickLeftNormalizedY < 0 OR G_Joystick.fJoystickLeftNormalizedY > 0 THEN
	G_Joystick.bJoystick4InUse := TRUE;
ELSE
	G_Joystick.bJoystick4InUse := FALSE;
END_IF

END_PROGRAM

// ---- ControlBox/FB_JoystickInputScaling.TcPOU
FUNCTION_BLOCK FB_JoystickInputScaling
VAR_INPUT
	bEnable  : BOOL;
	nRawInput : INT;
	stJoystickInputScaling : ST_JoystickInputScaling;
END_VAR
VAR_OUTPUT
	fNormalizedOutput : LREAL;
END_VAR
VAR
	fRawInput : LREAL;
	fTempInput : LREAL;
	fTempOutput : LREAL;
END_VAR

fRawInput := INT_TO_REAL(nRawInput);

fTempInput := fRawInput - stJoystickInputScaling.fNeutralInputValue;
IF fTempInput > stJoystickInputScaling.fNeutralDeadband THEN
	fTempOutput := fTempInput/(stJoystickInputScaling.fMaxInputValue - stJoystickInputScaling.fNeutralInputValue);
ELSIF fTempInput < -stJoystickInputScaling.fNeutralDeadband THEN
	fTempOutput := fTempInput/(stJoystickInputScaling.fNeutralInputValue - stJoystickInputScaling.fMinInputValue);
ELSE
	fTempOutput := 0;
END_IF

IF nRawInput = 0 THEN
	fNormalizedOutput := -0.0;
ELSIF NOT (bEnable) THEN
	fNormalizedOutput := -0.0;
ELSE 
	fNormalizedOutput := LIMIT(stJoystickInputScaling.fMinOutputValue, fTempOutput, stJoystickInputScaling.fMaxOutputValue);
END_IF

END_FUNCTION_BLOCK

// ---- ServoControl/P_ManualActuatorTest.TcPOU
PROGRAM P_ManualActuatorTest
VAR
	fbPathGenerator: FB_PathGenerator;
	Q1: BOOL;
	t: INT;
	ElapsedTime : LREAL;
	sinus :  LREAL;
	nsinus : UINT;
END_VAR

// This program is used only to make results for the manual controller. 
//Actuating each joint with sinusoidal wave and check the sensor


fbPathGenerator(bStart := G_Servo.bStartSinus, 
				TIN := T#15S , 
				Qout =>Q1, 
				t => ElapsedTime);
sinus := 70*SIN(ElapsedTime*2/2);
nsinus :=  LREAL_TO_UINT(sinus);

G_Servo.nServoPulseLenght1 := 350 ;// + sinus q1; 
G_Servo.nServoPulseLenght2 := 350;/// + sinus q3;			
G_Servo.nServoPulseLenght3 := 350; // Rotator
G_Servo.nServoPulseLenght4 := 350 + nsinus;// + nsinus;		
G_Servo.nServoPulseLenght6 := 350;

// Grasper
G_Servo.nServoPulseLenght5 := ButtonControlPulseLenght(fJoystickButtonFront := G_Buttons.bJoystickRightFrontEnable,
														fJoystickButtonBack := G_Buttons.bJoystickRightEnable,
															fNeutralPosition := 335);								
								
//Telescope using button					

														


				
(*

G_Servo.nServoPulseLenght6 := ButtonControlPulseLenght(fJoystickButtonFront := G_Buttons.bJoystickLeftEnable,
														fJoystickButtonBack := G_Buttons.bJoystickLeftFrontEnable,
														fNeutralPosition := 340);	

G_Servo.nServoPulseLenght1 := NormToPulseLenght(fJoyStickNormalized := G_Joystick.fJoystickLeftNormalizedX,
								fEndPulseLengthPositive := 390, fStartPulseLengthPositive := 368, fStartPulseLengthNegative := 333, fEndPulseLengthNegative := 310);

G_Servo.nServoPulseLenght2 := NormToPulseLenght(fJoyStickNormalized := G_Joystick.fJoystickLeftNormalizedY,
								fEndPulseLengthPositive := 410, fStartPulseLengthPositive := 360, fStartPulseLengthNegative := 340, fEndPulseLengthNegative := 290);								

G_Servo.nServoPulseLenght3 := NormToPulseLenght(fJoyStickNormalized := G_Joystick.fJoystickRightNormalizedX,
								fEndPulseLengthPositive := 410, fStartPulseLengthPositive := 360, fStartPulseLengthNegative := 340, fEndPulseLengthNegative := 290);								

G_Servo.nServoPulseLenght4 := NormToPulseLenght(fJoyStickNormalized := G_Joystick.fJoystickRightNormalizedY,
								fEndPulseLengthPositive := 410, fStartPulseLengthPositive := 360, fStartPulseLengthNegative := 340, fEndPulseLengthNegative := 290);									

								

														
														*)

END_PROGRAM

// ---- PathGenerator/FB_PathGenerator.TcPOU
FUNCTION_BLOCK FB_PathGenerator
VAR_INPUT
	bStart : BOOL;
	TIN : TIME;
END_VAR
VAR_OUTPUT
	Qout : BOOL; // Finished
	t : LREAL;
END_VAR
VAR
	tTimer : TON;
	tElappsed : TIME;
END_VAR

tTimer(IN := bStart, 
		PT := TIN,
		Q => Qout,
		ET => tElappsed);

t := TIME_TO_LREAL(tElappsed)/1000; // Time to S

END_FUNCTION_BLOCK

// ---- ServoControl/ButtonControlPulseLenght.TcPOU
FUNCTION ButtonControlPulseLenght : UINT
VAR_INPUT
	fJoystickButtonFront : BOOL;
	fJoystickButtonBack : BOOL;
	fNeutralPosition : LREAL;
END_VAR
VAR
	fActuation : LREAL;
	fservoPulseLenght : LREAL;
END_VAR

IF fJoystickButtonFront AND NOT(fJoystickButtonBack) THEN
	fActuation := -80;
ELSIF NOT(fJoystickButtonFront) AND fJoystickButtonBack THEN 
	fActuation := 80;
ELSE
	fActuation := 0;
END_IF

fservoPulseLenght := fActuation + fNeutralPosition;
ButtonControlPulseLenght := LREAL_TO_UINT(fservoPulseLenght);

END_FUNCTION

// ---- ServoControl/P_ManualControl.TcPOU
PROGRAM P_ManualControl
VAR
END_VAR


G_Servo.nServoPulseLenght1 := NormToPulseLenght(fJoyStickNormalized := G_Joystick.fJoystickLeftNormalizedX,
								fEndPulseLengthPositive := 390, fStartPulseLengthPositive := 368, fStartPulseLengthNegative := 333, fEndPulseLengthNegative := 310);

G_Servo.nServoPulseLenght2 := NormToPulseLenght(fJoyStickNormalized := G_Joystick.fJoystickLeftNormalizedY,
								fEndPulseLengthPositive := 410, fStartPulseLengthPositive := 360, fStartPulseLengthNegative := 340, fEndPulseLengthNegative := 290);								

G_Servo.nServoPulseLenght3 := NormToPulseLenght(fJoyStickNormalized := G_Joystick.fJoystickRightNormalizedX,
								fEndPulseLengthPositive := 410, fStartPulseLengthPositive := 370, fStartPulseLengthNegative := 350, fEndPulseLengthNegative := 290);								

G_Servo.nServoPulseLenght4 := NormToPulseLenght(fJoyStickNormalized := G_Joystick.fJoystickRightNormalizedY,
								fEndPulseLengthPositive := 410, fStartPulseLengthPositive := 360, fStartPulseLengthNegative := 340, fEndPulseLengthNegative := 290);									

								
// Grasper
G_Servo.nServoPulseLenght5 := ButtonControlPulseLenght(fJoystickButtonFront := G_Buttons.bJoystickRightFrontEnable,
														fJoystickButtonBack := G_Buttons.bJoystickRightEnable,
															fNeutralPosition := 325);								
								
//Telescope using button					
G_Servo.nServoPulseLenght6 := ButtonControlPulseLenght(fJoystickButtonFront := G_Buttons.bJoystickLeftEnable,
														fJoystickButtonBack := G_Buttons.bJoystickLeftFrontEnable,
														fNeutralPosition := 340);

END_PROGRAM

// ---- ServoControl/NormToPulseLenght.TcPOU
FUNCTION NormToPulseLenght : UINT
VAR_INPUT
	fJoystickNormalized : LREAL; // Signal from -1 to 1
	fEndPulseLengthPositive : LREAL; // Maximum pulse lenght for positive speed.
	fStartPulseLengthPositive : LREAL; // Minimum pulse lenght needed for starting movement in positive direction.
	fStartPulseLengthNegative : LREAL; // Pulse lenght needed for starting movement in positive direction.
	fEndPulseLengthNegative : LREAL; // Pulse lenght at maximum negative velocity.
END_VAR
VAR
	fservoPulseLenght : LREAL;
	fJoystickMultiplied : LREAL;
END_VAR

fJoystickMultiplied := (fEndPulseLengthPositive - fEndPulseLengthNegative)/2*fJoystickNormalized;


IF fJoystickNormalized > 0 THEN
	//Positive velocity
	fservoPulseLenght := fStartPulseLengthPositive + fJoystickMultiplied;
ELSIF fJoystickNormalized < 0 THEN
	// Negative velocity
	fservoPulseLenght := fStartPulseLengthNegative + fJoystickMultiplied;
ELSE
	//Idle
	fservoPulseLenght := (fStartPulseLengthNegative + fStartPulseLengthPositive)/2; 
END_IF



NormToPulseLenght := LREAL_TO_UINT(fservoPulseLenght);

END_FUNCTION

// ---- ActuatorLimits/P_ActuatorLimits.TcPOU
PROGRAM P_ActuatorLimits
VAR
	fbActuatorLimitsq1 : FB_ActuatorLimits;
	fbActuatorLimitsq2 : FB_ActuatorLimits;
	fbActuatorLimitsq3 : FB_ActuatorLimits;
	fbActuatorLimitsq4 : FB_ActuatorLimits;

END_VAR

fbActuatorLimitsq1(fsensorMinValue := G_ActuatorLimits.fq1Min,
					fsensorMaxValue := G_ActuatorLimits.fq1Max,
					fSensorSignal := G_SensorsScaled.q1,
					fServoSignalIn := G_Servo.f_u_q1,
					bMinReached => G_ActuatorLimits.bq1Min,
					bMaxReached => G_ActuatorLimits.bq1Max,
					fServoSignalOut => G_Servo.f_u_q1);


fbActuatorLimitsq2(fsensorMinValue := G_ActuatorLimits.fq2Min,
					fsensorMaxValue := G_ActuatorLimits.fq2Max,
					fSensorSignal := G_SensorsScaled.q2,
					fServoSignalIn := G_Servo.f_u_q2,
					bMinReached => G_ActuatorLimits.bq2Min,
					bMaxReached => G_ActuatorLimits.bq2Max,
					fServoSignalOut => G_Servo.f_u_q2);
					
					
fbActuatorLimitsq3(fsensorMinValue := G_ActuatorLimits.fq3Min,
					fsensorMaxValue := G_ActuatorLimits.fq3Max,
					fSensorSignal := G_SensorsScaled.q3,
					fServoSignalIn := G_Servo.f_u_q3,
					bMinReached => G_ActuatorLimits.bq3Min,
					bMaxReached => G_ActuatorLimits.bq3Max,
					fServoSignalOut => G_Servo.f_u_q3);
					
fbActuatorLimitsq4(fsensorMinValue := G_ActuatorLimits.fq4Min,
					fsensorMaxValue := G_ActuatorLimits.fq4Max,
					fSensorSignal := G_SensorsScaled.q4,
					fServoSignalIn := G_Servo.f_u_q4,
					bMinReached => G_ActuatorLimits.bq4Min,
					bMaxReached => G_ActuatorLimits.bq4Max,
					fServoSignalOut => G_Servo.f_u_q4);

END_PROGRAM

// ---- ActuatorLimits/FB_ActuatorLimits.TcPOU
FUNCTION_BLOCK FB_ActuatorLimits
VAR_INPUT
	fsensorMinValue : LREAL; //Sensor value at minimum actuator pos. OBS: G_Sensorscaled AFTER calibrating sensors!!!!!!
	fsensorMaxValue : LREAL; //Sensor value at minimum actuator pos. OBS: G_Sensorscaled AFTER calibrating sensors!!!!!!
	fSensorSignal : LREAL;
	fServoSignalIn : LREAL; // Signal out from controller. go trough this to prevent from running to end stop
END_VAR
VAR_OUTPUT
	bMinReached : BOOL;
	bMaxReached : BOOL;
	fServoSignalOut : LREAL;
END_VAR
VAR
END_VAR


IF fSensorSignal <= fsensorMinValue THEN
	bMinReached := TRUE;
	// Peventing from running in wrong direction when closee to end stop:
	IF fServoSignalIn <= 0 THEN
		fServoSignalOut := 0;
	ELSE
		fServoSignalOut := fServoSignalIn;
	END_IF
ELSIF fSensorSignal >= fsensorMaxValue THEN
	bMaxReached := TRUE;
	// Peventing from running in wrong direction when closee to end stop:
	IF fServoSignalIn >= 0 THEN
		fServoSignalOut := 0;
	ELSE
		fServoSignalOut := fServoSignalIn;
	END_IF
ELSE
	bMinReached := FALSE;
	bMaxReached := FALSE;
	fServoSignalOut := fServoSignalIn;
END_IF

END_FUNCTION_BLOCK

// ---- PathGenerator/P_PathGeneration_2.TcPOU
PROGRAM P_PathGeneration_2
VAR
	fbPathGenerator : FB_PathGenerator;
	Q1 : BOOL;
	ElapsedTime : LREAL;
	TimeX : LREAL := 2.5;
	TimeY : LREAL := 1.2;
	TimeZ : LREAL := 1.2;
	TimeEachSequence: INT;
	cartesianVelocity : LREAL;
	timescaling: LREAL;
END_VAR

// FOR  TELESCOPE TUNING
timescaling := 3;
cartesianVelocity := 0.050/timescaling; // OPEN LOOP: Very much difference between m/s

fbPathGenerator(bStart := G_Path.bStartPath, 
				TIN := T#150S , 
				Qout =>Q1, 
				t => ElapsedTime);


IF ElapsedTime>= 0*timescaling AND ElapsedTime< 2*timescaling AND G_Path.bStartPath THEN 
	G_Path.bPathRunning := TRUE;
	G_Path.bPathFinnish := FALSE;
	G_InverseKinematics.fvXref := cartesianVelocity; //mm/S
	G_InverseKinematics.fvYref := 0; //mm/S
	G_InverseKinematics.fvZref := 0; //mm/S
(*ELSIF ElapsedTime = 2*timescaling THEN
	G_Toolpoint.fXref := G_Toolpoint.fX; // RESET PATH TO CURRENT PATH IN TRANSITIONS
	G_Toolpoint.fYref := G_Toolpoint.fY;
	G_Toolpoint.fZref := G_Toolpoint.fZ;*)
ELSIF ElapsedTime>= 2*timescaling AND ElapsedTime < 4*timescaling THEN
	G_InverseKinematics.fvXref := 0; //mm/S
	G_InverseKinematics.fvYref := cartesianVelocity; //mm/S
	G_InverseKinematics.fvZref := 0; //mm/S
(*ELSIF ElapsedTime = 4*timescaling THEN
	G_Toolpoint.fXref := G_Toolpoint.fX; // RESET PATH TO CURRENT PATH IN TRANSITIONS
	G_Toolpoint.fYref := G_Toolpoint.fY;
	G_Toolpoint.fZref := G_Toolpoint.fZ;*)
ELSIF ElapsedTime>= 4*timescaling AND ElapsedTime < 6*timescaling THEN
	G_InverseKinematics.fvXref := 0; //mm/S
	G_InverseKinematics.fvYref := 0; //mm/S
	G_InverseKinematics.fvZref := cartesianVelocity; //mm/S
(*ELSIF ElapsedTime = 6*timescaling THEN
	G_Toolpoint.fXref := G_Toolpoint.fX; // RESET PATH TO CURRENT PATH IN TRANSITIONS
	G_Toolpoint.fYref := G_Toolpoint.fY;
	G_Toolpoint.fZref := G_Toolpoint.fZ;*)
ELSIF ElapsedTime>= 6*timescaling AND ElapsedTime < 8*timescaling THEN
	G_InverseKinematics.fvXref := cartesianVelocity; //mm/S
	G_InverseKinematics.fvYref := -cartesianVelocity; //mm/S
	G_InverseKinematics.fvZref := 0; //mm/S
(*ELSIF ElapsedTime = 8*timescaling THEN
	G_Toolpoint.fXref := G_Toolpoint.fX; // RESET PATH TO CURRENT PATH IN TRANSITIONS
	G_Toolpoint.fYref := G_Toolpoint.fY;
	G_Toolpoint.fZref := G_Toolpoint.fZ;*)
ELSIF ElapsedTime>= 8*timescaling AND ElapsedTime < 13*timescaling THEN
	G_InverseKinematics.fvXref := 0; //mm/S
	G_InverseKinematics.fvYref := cartesianVelocity; //mm/S
	G_InverseKinematics.fvZref := 0; //mm/S
(*ELSIF ElapsedTime = 13*timescaling THEN
	G_Toolpoint.fXref := G_Toolpoint.fX; // RESET PATH TO CURRENT PATH IN TRANSITIONS
	G_Toolpoint.fYref := G_Toolpoint.fY;
	G_Toolpoint.fZref := G_Toolpoint.fZ;*)
ELSIF ElapsedTime>= 13*timescaling AND ElapsedTime < 17*timescaling THEN
	G_InverseKinematics.fvXref := -cartesianVelocity; //mm/S
	G_InverseKinematics.fvYref := -cartesianVelocity; //mm/S
	G_InverseKinematics.fvZref := 0; //mm/S
(*ELSIF ElapsedTime = 17*timescaling THEN
	G_Toolpoint.fXref := G_Toolpoint.fX; // RESET PATH TO CURRENT PATH IN TRANSITIONS
	G_Toolpoint.fYref := G_Toolpoint.fY;
	G_Toolpoint.fZref := G_Toolpoint.fZ;*)
ELSIF ElapsedTime>= 17*timescaling AND ElapsedTime < 18.5*timescaling THEN
	G_InverseKinematics.fvXref := 0; //mm/S
	G_InverseKinematics.fvYref := 0; //mm/S
	G_InverseKinematics.fvZref := -cartesianVelocity; //mm/S
ELSIF ElapsedTime>= 18.5*timescaling AND ElapsedTime < 19.5*timescaling THEN
	G_InverseKinematics.fvXref := 0; //mm/S
	G_InverseKinematics.fvYref := -cartesianVelocity; //mm/S
	G_InverseKinematics.fvZref := 0; //mm/S
ELSE
	G_Path.bPathRunning := FALSE;
	G_Path.bPathFinnish := TRUE;
	G_Path.bStartPath := FALSE;
	ElapsedTime := 0;
	G_InverseKinematics.fvXref := 0; //mm/S
	G_InverseKinematics.fvYref := 0; //mm/S
	G_InverseKinematics.fvZref := 0; //mm/S
END_IF



(*
CASE CaseInt OF

1:  
fbPathGenerator(bStart := G_Path.bStartPath,
TIN := T#2S, 
Coordinate => G_InverseVelocityKinematics.fvXref, 
Qout => Q1);
IF Q1 THEN
	CaseInt:=2;
END_IF


2:     
fbPathGenerator2(bStart := G_Path.bStartPath,
TIN := T#2S, 
Coordinate => G_InverseVelocityKinematics.fvYref, 
Qout => Q2);
IF Q2 THEN
	CaseInt:=3;
END_IF

3:     
fbPathGenerator3(bStart := G_Path.bStartPath,
TIN := T#2S, 
Coordinate => G_InverseVelocityKinematics.fvZref, 
Qout => Q3);
IF Q3 THEN
	G_Path.bStartPath := FALSE;
	CaseInt:=1;
	Q1 := FALSE;
	Q2 := FALSE;
	Q3 := FALSE;
END_IF

END_CASE;

*)

END_PROGRAM

// ---- Kinematics_CraneFrame/P_CartesianVelFromJoystick.TcPOU
PROGRAM P_CartesianVelFromJoystick
VAR

	fbJoystickToCartesianVelocity1 : FB_JoystickToCartesianVelocity;
	fbJoystickToCartesianVelocity2 : FB_JoystickToCartesianVelocity;
	fbJoystickToCartesianVelocity3 : FB_JoystickToCartesianVelocity;
END_VAR

						
// Mapping joistick to cartesian linear velocity
fbJoystickToCartesianVelocity1(fNormalizezJoistick := G_Joystick.fJoystickLeftNormalizedY,
								fScalingFactor := 0.02, //Corresponding to linear velocity toolpoint in m/s
								fAxisVelocity => G_InverseKinematics.fvXref);
								
fbJoystickToCartesianVelocity2(fNormalizezJoistick := G_Joystick.fJoystickLeftNormalizedX,
								fScalingFactor := 0.02,
								fAxisVelocity => G_InverseKinematics.fvYref);

fbJoystickToCartesianVelocity3(fNormalizezJoistick := -G_Joystick.fJoystickRightNormalizedY, // Direction on the joystick inverted
								fScalingFactor := 0.02,
								fAxisVelocity => G_InverseKinematics.fvZref);

END_PROGRAM

// ---- JoystickToCartesianVelocity/FB_JoystickToCartesianVelocity.TcPOU
FUNCTION_BLOCK FB_JoystickToCartesianVelocity
VAR_INPUT
	fNormalizezJoistick : LREAL;
	fScalingFactor : LREAL; 
END_VAR
VAR_OUTPUT
	fAxisVelocity : LREAL;
END_VAR
VAR
END_VAR



fAxisVelocity := fNormalizezJoistick*fScalingFactor;

END_FUNCTION_BLOCK

// ---- ActuatorLimits/P_CartesianLimit.TcPOU
PROGRAM P_CartesianLimit
VAR
	fbXLIMIT : FB_CartesianVelLimit;
	fbYLIMIT : FB_CartesianVelLimit;
	fbZLIMIT : FB_CartesianVelLimit;
END_VAR

fbXLIMIT(axisVelocityIn := G_InverseKinematics.fvXref,
							axisPosition := G_Toolpoint.fX,
							axisMinPosition := G_ActuatorLimits.fXMin,
							axisMaxPosition := G_ActuatorLimits.fXMax,
							axisVelocityOut => G_InverseKinematics.fvXref);


fbXLIMIT(axisVelocityIn := G_InverseKinematics.fvYref,
							axisPosition := G_Toolpoint.fY,
							axisMinPosition := G_ActuatorLimits.fYMin,
							axisMaxPosition := G_ActuatorLimits.fYMax,
							axisVelocityOut => G_InverseKinematics.fvYref);

fbXLIMIT(axisVelocityIn := G_InverseKinematics.fvZref,
							axisPosition := G_Toolpoint.fZ,
							axisMinPosition := G_ActuatorLimits.fZMin,
							axisMaxPosition := G_ActuatorLimits.fZMax,
							axisVelocityOut => G_InverseKinematics.fvZref);

END_PROGRAM

// ---- ActuatorLimits/FB_CartesianVelLimit.TcPOU
FUNCTION_BLOCK FB_CartesianVelLimit
VAR_INPUT
	axisVelocityIn : LREAL;
	axisPosition : LREAL;
	axisMinPosition : LREAL;
	axisMaxPosition : LREAL;
END_VAR
VAR_OUTPUT
	axisVelocityOut : LREAL;
END_VAR
VAR
END_VAR

IF axisPosition >= axisMaxPosition THEN
	//Max reached
	IF axisVelocityIn >= 0 THEN
		axisVelocityOut := 0;
	ELSE
		axisVelocityOut := axisVelocityIn;
	END_IF
ELSIF axisPosition <= axisMinPosition THEN
	//Min reached
	IF axisVelocityIn <= 0 THEN
		axisVelocityOut := 0;
	ELSE
		axisVelocityOut := axisVelocityIn;
	END_IF
ELSE
	// None reached
axisVelocityOut := axisVelocityIn;
END_IF

END_FUNCTION_BLOCK

// ---- HeaveCompensation/P_Heave.TcPOU
PROGRAM P_Heave
VAR
	fbGet3r : FB_Get3r;
	fbGenr1b : FB_Genr1b;
	fbToolpointPositionIntegrator2 : FB_ToolpointPositionIntegrator;
	thethaThreshold : LREAL := 0.5; //Degrees
END_VAR

//  Remove offset from tipping angle
G_Heave.fTheta := G_SensorInput.fYRotDeg - G_Heave.fThetaStart;

// Tune threshold
thethaThreshold := 0.3;


//Set angle threshold due to physical limitations
IF G_Heave.fTheta < 0 THEN
	G_Heave.fTheta := 0;
ELSIF G_Heave.fTheta > 13 THEN
	G_Heave.fTheta := 13; //Degrees
END_IF


	


// Check if tilting is active:
IF G_Heave.fTheta > thethaThreshold AND G_Heave.fTheta < 13 THEN
	//CODE FOR HEAVE COMPENSATION
//integrating r3 to include tolpoint velocity. r3 frame coordinate is paralell to crane coordinate with theta = 0 
fbToolpointPositionIntegrator2(fXref :=G_Heave.r3x,
									fYref :=G_Heave.r3y,
									fZref := G_Heave.r3z,
								fXrefOut => G_Heave.r3x,
								fYrefOut => G_Heave.r3y,
								fZrefOut => G_Heave.r3z);


// Generate vector from crane base to toolpoint in crane coordinate, based on the r3 vector in crane coordinate
fbGenr1b(thetaDeg := G_Heave.fTheta,
			r3x := G_Heave.r3x,
			r3y := G_Heave.r3y,
			r3z := G_Heave.r3z,
			r1bx => G_Heave.r1bxCrane,
			r1by => G_Heave.r1byCrane,
			r1bz => G_Heave.r1bzCrane);

// Writing the desired position coordinate in crane frame
G_Toolpoint.fXref := G_Heave.r1bxCrane;
G_Toolpoint.fYref := G_Heave.r1byCrane;
G_Toolpoint.fZref := G_Heave.r1bzCrane;


ELSE
	//CODE FOR SETTING r3 when angle is approx 0
	fbGet3r(xToolpointCraneFrame := G_Toolpoint.fXref,  // Use ref here so the r3 vector gets updated in cartesian control aswell
			yToolpointCraneFrame := G_Toolpoint.fYref,
			zToolpointCraneFrame := G_Toolpoint.fZref,
			r3x => G_Heave.r3x,
			r3y => G_Heave.r3y,
			r3z => G_Heave.r3z);
			
	P_VelToPos();			
END_IF

END_PROGRAM

// ---- HeaveCompensation/FB_Get3r.TcPOU
FUNCTION_BLOCK FB_Get3r
VAR_INPUT
    xToolpointCraneFrame: LREAL; //m
    yToolpointCraneFrame: LREAL; //m
    zToolpointCraneFrame: LREAL; //m
END_VAR
VAR_OUTPUT
    r3x: LREAL; //m
    r3y: LREAL; //m
    r3z: LREAL; //m
END_VAR

(* Outport: '<Root>/r3x' incorporates:
 *  MATLAB Function: '<Root>/MATLAB Function1' *)
(* CraneFrame toolpoint *)
(* MATLAB Function 'MATLAB Function1': '<S1>:1' *)
(* '<S1>:1:4' r1a = [xToolpointCraneFrame; *)
(* '<S1>:1:5'    yToolpointCraneFrame ; *)
(* '<S1>:1:6'     zToolpointCraneFrame]; *)
(* Vector from tippingpoint to crane *)
(* '<S1>:1:9' r2a = [-37;%mm *)
(* '<S1>:1:10'     0; *)
(* '<S1>:1:11'     10]; *)
(* mm *)
(* mm *)
(* '<S1>:1:13' r3 = r1a + r2a; *)
(* '<S1>:1:14' r3x = r3(1); *)
(* '<S1>:1:15' r3y = r3(2); *)
(* '<S1>:1:16' r3z = r3(3); *)
r3x := xToolpointCraneFrame -0.037;
(* Outport: '<Root>/r3y' incorporates:
 *  MATLAB Function: '<Root>/MATLAB Function1' *)
r3y := yToolpointCraneFrame;
(* Outport: '<Root>/r3z' incorporates:
 *  MATLAB Function: '<Root>/MATLAB Function1' *)
r3z := zToolpointCraneFrame + 0.013;

END_FUNCTION_BLOCK

// ---- HeaveCompensation/FB_Genr1b.TcPOU
FUNCTION_BLOCK FB_Genr1b
VAR_INPUT
    thetaDeg: LREAL;
    r3x: LREAL; //m
    r3y: LREAL; //m
    r3z: LREAL; //m
END_VAR
VAR_OUTPUT
    r1bx: LREAL; //m
    r1by: LREAL; //m
    r1bz: LREAL; //m
END_VAR
VAR_TEMP
    theta: LREAL;
    r1b_crane: ARRAY [0..2] OF LREAL;
    r1b_crane_tmp: LREAL;
    r1b_crane_tmp_0: LREAL;
    r1b_crane_tmp_1: LREAL;
    r1b_crane_tmp_2: LREAL;
    r1b_crane_tmp_3: ARRAY [0..8] OF LREAL;
    r1b_crane_tmp_4: ARRAY [0..2] OF LREAL;
    i: DINT;
END_VAR

(* MATLAB Function: '<Root>/MATLAB Function2' *)
(* Vector from tippingpoint to crane *)
(* MATLAB Function 'MATLAB Function2': '<S1>:1' *)
(* '<S1>:1:4' r2a = [-37;0;10]; *)
(* mm *)
(* '<S1>:1:6' r3 = [r3x,r3y,r3z]'; *)
(* '<S1>:1:7' theta = deg2rad(thetaDeg); *)
theta := 0.017453292519943295 * thetaDeg;
(* RotationAroundYAxis *)
(* '<S1>:1:10' Arot = ArotY(theta); *)
(* Returns the rotation matrix around y axis for given theta input *)
(* 'ArotY:3' Arot = [ cos(theta) 0 sin(theta); *)
(* 'ArotY:4'             0        1      0; *)
(* 'ArotY:5'     -sin(theta)     0   cos(theta)]; *)
(* '<S1>:1:11' AnegRot = ArotY(-theta); *)
(* Returns the rotation matrix around y axis for given theta input *)
(* 'ArotY:3' Arot = [ cos(theta) 0 sin(theta); *)
(* 'ArotY:4'             0        1      0; *)
(* 'ArotY:5'     -sin(theta)     0   cos(theta)]; *)
(* New vectors after rot *)
(* '<S1>:1:14' r2b = Arot*r2a; *)
(* r2 new in frame coordinate *)
(* '<S1>:1:15' r1b = r3-r2b; *)
(* r1b new in frame coordinate *)
(* '<S1>:1:16' r1b_crane = AnegRot*r1b; *)
r1b_crane_tmp := SIN( -theta);
r1b_crane_tmp_0 := COS( -theta);
r1b_crane_tmp_1 := SIN(theta);
r1b_crane_tmp_2 := COS(theta);
(* MATLAB Function: '<Root>/MATLAB Function2' *)
r1b_crane_tmp_3[0] := r1b_crane_tmp_2;
r1b_crane_tmp_3[3] := 0.0;
r1b_crane_tmp_3[6] := r1b_crane_tmp_1;
r1b_crane_tmp_3[1] := 0.0;
r1b_crane_tmp_3[4] := 1.0;
r1b_crane_tmp_3[7] := 0.0;
r1b_crane_tmp_3[2] :=  -r1b_crane_tmp_1;
r1b_crane_tmp_3[5] := 0.0;
r1b_crane_tmp_3[8] := r1b_crane_tmp_2;
(* MATLAB Function: '<Root>/MATLAB Function2' *)
FOR i := 0 TO 2 DO 
    r1b_crane_tmp_4[i] := (r1b_crane_tmp_3[i + 6] * 0.013) + (r1b_crane_tmp_3[i] * -0.037);
END_FOR;
(* MATLAB Function: '<Root>/MATLAB Function2' *)
r1b_crane_tmp_3[0] := r1b_crane_tmp_0;
r1b_crane_tmp_3[3] := 0.0;
r1b_crane_tmp_3[6] := r1b_crane_tmp;
r1b_crane_tmp_3[2] :=  -r1b_crane_tmp;
r1b_crane_tmp_3[5] := 0.0;
r1b_crane_tmp_3[8] := r1b_crane_tmp_0;
r1b_crane_tmp_3[1] := 0.0;
r1b_crane_tmp := r3x - r1b_crane_tmp_4[0];
r1b_crane_tmp_3[4] := 1.0;
r1b_crane_tmp_0 := r3y - r1b_crane_tmp_4[1];
r1b_crane_tmp_3[7] := 0.0;
r1b_crane_tmp_1 := r3z - r1b_crane_tmp_4[2];
(* MATLAB Function: '<Root>/MATLAB Function2' *)
FOR i := 0 TO 2 DO 
    r1b_crane[i] := (r1b_crane_tmp_3[i + 6] * r1b_crane_tmp_1) + ((r1b_crane_tmp_3[i + 3] * r1b_crane_tmp_0) + (r1b_crane_tmp_3[i] * r1b_crane_tmp));
END_FOR;
(* Outport: '<Root>/r1bx' incorporates:
 *  MATLAB Function: '<Root>/MATLAB Function2' *)
(* r1b new in crane coordinate *)
(* '<S1>:1:19' r1bx = r1b_crane(1); *)
(* '<S1>:1:20' r1by = r1b_crane(2); *)
(* '<S1>:1:21' r1bz = r1b_crane(3); *)
r1bx := r1b_crane[0];
(* Outport: '<Root>/r1by' incorporates:
 *  MATLAB Function: '<Root>/MATLAB Function2' *)
r1by := r1b_crane[1];
(* Outport: '<Root>/r1bz' incorporates:
 *  MATLAB Function: '<Root>/MATLAB Function2' *)
r1bz := r1b_crane[2];

END_FUNCTION_BLOCK

// ---- Kinematics_CraneFrame/FB_ToolpointPositionIntegrator.TcPOU
FUNCTION_BLOCK FB_ToolpointPositionIntegrator
VAR_INPUT
	fXref : LREAL;
	fYref : LREAL;
	fZref : LREAL;
END_VAR
VAR_OUTPUT
	fXrefOut : LREAL;
	fYrefOut : LREAL;
	fZrefOut : LREAL;
END_VAR
VAR
		cycleTime : LREAL :=  0.01; //s
END_VAR

fXrefOut := fXref;


IF G_Path.bStartPath OR G_Joystick.bJoystick2InUse OR G_Joystick.bJoystick4InUse OR G_Joystick.bJoystick3InUse OR G_Heave.bHeaveActive  THEN
	fXrefOut := fXref;
	fYrefOut := fYref;
	fZrefOut := fZref;
	fXrefOut := fXrefOut + G_InverseKinematics.fvXref * cycleTime;
	fYrefOut := fYrefOut + G_InverseKinematics.fvYref * cycleTime;
	fZrefOut := fZrefOut + G_InverseKinematics.fvZref * cycleTime;
ELSE
	fXrefOut := G_Toolpoint.fX;
	fYrefOut := G_Toolpoint.fY;
	fZrefOut := G_Toolpoint.fZ;
END_IF

END_FUNCTION_BLOCK

// ---- ServoControl/P_VelToPos.TcPOU
PROGRAM P_VelToPos
VAR
		fbToolpointPositionIntegrator : FB_ToolpointPositionIntegrator;
END_VAR

fbToolpointPositionIntegrator(fXref := G_Toolpoint.fXref,
								fYref := G_Toolpoint.fYref,
								fZref := G_Toolpoint.fZref,
								fXrefOut => G_Toolpoint.fXref,
								fYrefOut => G_Toolpoint.fYref,
								fZrefOut => G_Toolpoint.fZref);

END_PROGRAM

// ---- ServoControl/P_CartesianController.TcPOU
PROGRAM P_CartesianController
VAR
	fbPIDController : FB_PID_Controller;
	fbInverseKinematics : FB_InverseKinematics;
END_VAR



fbInverseKinematics(q1Inn := G_SensorsScaled.q1,// Inverse kinematics
					q2Inn := G_SensorsScaled.q2,
					q3Inn := G_SensorsScaled.q3,
					q4Inn := G_SensorsScaled.q4,
					r1bx := G_ToolPoint.fXref,    // Possibly change for r1bx???
					r1by := G_ToolPoint.fYref,
					r1bz := G_ToolPoint.fZref,
					Vx := G_InverseKinematics.fvXref,
					Vy := G_InverseKinematics.fvYref,
					Vz := G_InverseKinematics.fvZref,
					q1 => G_InverseKinematics.f_q1_ref,
					q2 => G_InverseKinematics.f_q2_ref,
					q3 => G_InverseKinematics.f_q3_ref,
					q4Dot => G_InverseKinematics.fq4Dotref,
					success => G_InverseKinematics.bKinematicsSucsessful);

P_NormalizeJointVel(); // Joint vel to normalized for telescope

fbPIDController(); // P controller

P_ActuatorLimits(); // Checking sensors and light lamps in HMI, and preventing automode from chrashing actuators. Called after PID, before actuation

P_CarteseanControllerServoActuation4DOF();	// Servo actuation

END_PROGRAM

// ---- ServoControl/FB_PID_Controller.TcPOU
FUNCTION_BLOCK FB_PID_Controller
VAR_INPUT
END_VAR
VAR_OUTPUT
END_VAR
VAR
	// Position Gains
	Kp1 : LREAL;
	Kp2 : LREAL;
	Kp3 : LREAL;
	Ki1 : LREAL;
	Ki2 : LREAL;
	Ki3 : LREAL;
	Kd1 : LREAL;
	Kd2 : LREAL;
	Kd3 : LREAL;
	
	
	
	// FF GAINS
	KF4 : LREAL;
	FFPart4 : LREAL;
	FFPart4_B : LREAL;

	pid1 : FB_PID;
	pid2 : FB_PID;
	pid3 : FB_PID;
	
END_VAR


KF4 := 0.05; // FF PART

(*
// Position Gains
Kp1 := 5;
Kp2 := 8;
Kp3 := 6;
Ki1 := 1;
Ki2 := 1;
Ki3 := 1;
Kd1 := 0.05;
Kd2 := 0.05;
Kd3 := 0.05;
*)

Kp1 := 5;
Kp2 := 8;
Kp3 := 6;
Ki1 := 1;
Ki2 := 1;
Ki3 := 1;
Kd1 := 0.05;
Kd2 := 0.05;
Kd3 := 0.05;




FFPart4 := KF4*G_Servo.fNormalizedActuatorVelFeedForward_q4Dot;



// Favorizing return of the telescope
IF FFPart4 <= 0 THEN
	FFPart4_B := FFPart4*10;
ELSE
	FFPart4_B := FFPart4;
END_IF


G_Servo.f_u_q4 := FFPart4_B;    // FF


// Closed loop control joint q1
pid1(SetPoint :=  G_InverseKinematics.f_q1_ref,
		SensorValue := G_SensorsScaled.q1,
		Kp := Kp1,
		Ki := Ki1,
		Kd := Kd1,
		MaxOutput := 1,
		MinOutput := -1,
		ResetIntegral := TRUE,
		Output => G_Servo.f_u_q1);

// Closed loop control joint q2
pid2(SetPoint :=  G_InverseKinematics.f_q2_ref,
		SensorValue := G_SensorsScaled.q2,
		Kp := Kp2,
		Ki := Ki2,
		Kd := Kd2,
		MaxOutput := 1,
		MinOutput := -1,
		ResetIntegral := TRUE,
		Output => G_Servo.f_u_q2);
		
// Closed loop control joint q3		
pid3(SetPoint :=  G_InverseKinematics.f_q3_ref,
		SensorValue := G_SensorsScaled.q3,
		Kp := Kp3,
		Ki := Ki3,
		Kd := Kd3,
		MaxOutput := 1,
		MinOutput := -1,
		ResetIntegral := TRUE,
		Output => G_Servo.f_u_q3);

END_FUNCTION_BLOCK

// ---- ServoControl/FB_PID.TcPOU
FUNCTION_BLOCK FB_PID
VAR_INPUT
    SetPoint : LREAL;               
    SensorValue : LREAL;        
    Kp : LREAL;                     
    Ki : LREAL;                     
    Kd : LREAL;                     
    MaxOutput : LREAL;              
    MinOutput : LREAL; 
	ResetIntegral : BOOL;             
END_VAR
VAR_OUTPUT
    Output : LREAL;                 
END_VAR
VAR
    Error : LREAL;                 
    Integral : LREAL;               
    LastError : LREAL := 0.0;       
    Derivative : LREAL;             
    timestep : LREAL := 0.01;            
END_VAR


IF ResetIntegral THEN
	Integral := 0.0;
	ResetIntegral := FALSE;
END_IF


Error := Setpoint - SensorValue;


Integral := Integral + (Error * timestep);


IF Integral > MaxOutput THEN
	Integral := MaxOutput;
ELSIF Integral < MinOutput THEN
    Integral := MinOutput;
END_IF;

Derivative := (Error - LastError) / timestep;

LastError := Error;

Output := (Kp * Error) + (Ki * Integral) + (Kd * Derivative);

IF Output > MaxOutput THEN
	Output := MaxOutput;
ELSIF Output < MinOutput THEN
	Output := MinOutput;
END_IF;

END_FUNCTION_BLOCK

// ---- KinematicsForwAndInverseMatLab/FB_InverseKinematics.TcPOU
FUNCTION_BLOCK FB_InverseKinematics
VAR_INPUT
    q1Inn: LREAL;
    q2Inn: LREAL;
    q3Inn: LREAL;
    q4Inn: LREAL;
    r1bx: LREAL;
    r1by: LREAL;
    r1bz: LREAL;
    Vx: LREAL;
    Vy: LREAL;
    Vz: LREAL;
END_VAR
VAR_OUTPUT
    q1: LREAL;
    q2: LREAL;
    q3: LREAL;
    q4Dot: LREAL;
    success: BOOL;
END_VAR
VAR
    f: ARRAY [0..5] OF SINT := [0,0,1,0,0,0];
    g: ARRAY [0..5] OF LREAL := [0.0,1.0,0.0,-0.1569,0.0,-0.02745];
    h: ARRAY [0..5] OF LREAL := [0.0,1.0,0.0,-0.1569,0.0,0.15197];
    p_a: ARRAY [0..8] OF SINT := [1,0,0,0,1,0,0,0,1];
    b_l: ARRAY [0..5] OF SINT := [0,0,0,1,0,0];
    i0_MatrixLog3: MatrixLog3;
    i0_eye: eye;
    i0_pinv: pinv;
    i0_pinv_i: pinv_i;
END_VAR
VAR_TEMP
    q5Inn: LREAL;
    S5: ARRAY [0..5] OF LREAL;
    S6: ARRAY [0..5] OF LREAL;
    J: ARRAY [0..35] OF LREAL;
    Slist: ARRAY [0..29] OF LREAL;
    M: ARRAY [0..15] OF LREAL;
    T: ARRAY [0..15] OF LREAL;
    thetalist0: ARRAY [0..4] OF LREAL;
    Tsb: ARRAY [0..15] OF LREAL;
    Vs: ARRAY [0..5] OF LREAL;
    err: BOOL;
    b_i: DINT;
    c_i: DINT;
    theta: LREAL;
    Js: ARRAY [0..29] OF LREAL;
    d_i: DINT;
    e_i: DINT;
    b_theta: LREAL;
    se3mat: ARRAY [0..15] OF LREAL;
    omgtheta: ARRAY [0..2] OF LREAL;
    omgmat: ARRAY [0..8] OF LREAL;
    a: ARRAY [0..15] OF LREAL;
    g_a: LREAL;
    V: ARRAY [0..5] OF LREAL;
    b_R: ARRAY [0..8] OF LREAL;
    b_omgmat: ARRAY [0..8] OF LREAL;
    l_a: LREAL;
    d_theta: LREAL;
    Slist_tmp: ARRAY [0..5] OF SINT;
    g_theta: LREAL;
    e_theta: LREAL;
    h_theta: LREAL;
    j_theta: LREAL;
    i: DINT;
    thetalist0_0: LREAL;
    se3mat_0: ARRAY [0..2] OF LREAL;
    a_0: ARRAY [0..15] OF LREAL;
    tmp: ARRAY [0..8] OF LREAL;
    Tsb_0: ARRAY [0..35] OF LREAL;
    tmp_0: ARRAY [0..8] OF LREAL;
    tmp_1: ARRAY [0..29] OF LREAL;
    tmp_2: ARRAY [0..5] OF LREAL;
    b_T: ARRAY [0..15] OF LREAL;
    tmp_3: ARRAY [0..8] OF LREAL;
    tmp_4: ARRAY [0..8] OF LREAL;
    T_0: ARRAY [0..35] OF LREAL;
    tmp_5: ARRAY [0..8] OF LREAL;
    Slist_tmp_0: DINT;
    a_tmp_tmp: DINT;
    omgmat_tmp: DINT;
    x_tmp: LREAL;
    R_tmp: DINT;
    c_theta: LREAL;
    f_theta: LREAL;
    i_theta: LREAL;
END_VAR

(* MATLAB Function: '<Root>/MATLAB Function3' *)
(* SIMPLIYFIED 3 DOF *)
(* MATLAB Function 'MATLAB Function3': '<S1>:1' *)
(* '<S1>:1:4' q5Inn = -(q2Inn+q3Inn); *)
q5Inn :=  -(q2Inn + q3Inn);
(* ALWAYS HORISONTAL DUMMY JOINT *)
(* '<S1>:1:5' q6Inn = -q1Inn; *)
(* ALWAYS PARRALELL TO ORGIN *)
(* Lenght from assy drawing *)
(* '<S1>:1:8' l1 = 156.9/1000; *)
(* m *)
(* '<S1>:1:9' l2 = 27.45/1000; *)
(* m *)
(* '<S1>:1:10' l3 = 179.42/1000; *)
(* m *)
(* '<S1>:1:11' l4 = 26.86/1000; *)
(* m *)
(* From Telescope drawing (IN assy drawing) *)
(* l5 = 163.43;  *)
(* '<S1>:1:17' l5 = 167.25/1000; *)
(* m Corrected after sensor calibration  *)
(* '<S1>:1:18' l6 = 1.75/1000; *)
(* m *)
(* '<S1>:1:19' W1 = -l2+l3+l5+q4Inn; *)
(* '<S1>:1:20' W2 = l4; *)
(* '<S1>:1:21' W3 = l1-l6; *)
(* Position of each joint *)
(* '<S1>:1:25' a1 = [0; 0; 0]; *)
(* '<S1>:1:26' a2 = [-l2; 0; l1]; *)
(* '<S1>:1:27' a3 = [-l2+l3; 0; l1]; *)
(* '<S1>:1:28' a5 = [W1; W2; W3]; *)
(* '<S1>:1:29' a6 = [W1; W2; W3]; *)
(* Screw axis of ech joint *)
(* '<S1>:1:32' Sw1 = [0; 0; 1]; *)
(* '<S1>:1:33' Sw2 = [0; 1; 0]; *)
(* '<S1>:1:34' Sw3 = [0; 1; 0]; *)
(* '<S1>:1:35' Sw5 = [0; 1; 0]; *)
(* '<S1>:1:36' Sw6 = [0; 0; 1]; *)
(* '<S1>:1:38' Sv1 = cross(a1,Sw1); *)
(* '<S1>:1:39' Sv2 = cross(a2,Sw2); *)
(* '<S1>:1:40' Sv3 = cross(a3,Sw3); *)
(* '<S1>:1:41' Sv5 = cross(a5,Sw5); *)
(* '<S1>:1:42' Sv6 = cross(a6,Sw6); *)
(* '<S1>:1:44' S1 = [Sw1;Sv1]; *)
(* '<S1>:1:45' S2 = [Sw2;Sv2]; *)
(* '<S1>:1:46' S3 = [Sw3;Sv3]; *)
(* '<S1>:1:47' S4 = [0;0;0;1;0;0]; *)
(* '<S1>:1:48' S5 = [Sw5;Sv5]; *)
S5[3] := -0.15515;
S5[4] := 0.0;
S5[5] := q4Inn + 0.31922;
(* '<S1>:1:49' S6 = [Sw6;Sv6]; *)
S5[0] := 0.0;
S6[0] := 0.0;
S5[1] := 1.0;
S6[1] := 0.0;
S5[2] := 0.0;
S6[2] := 1.0;
S6[3] := 0.02686;
S6[4] := 0.0 - (q4Inn + 0.31922);
S6[5] := 0.0;
(* '<S1>:1:51' M = [[1 0 0 W1]; *)
(* '<S1>:1:52'     [0 1 0 W2]; *)
(* '<S1>:1:53'     [0 0 1 W3]; *)
(* '<S1>:1:54'     [0 0 0 1];]; *)
(* MATLAB Function: '<Root>/MATLAB Function3' *)
M[0] := 1.0;
M[4] := 0.0;
M[8] := 0.0;
M[12] := q4Inn + 0.31922;
M[1] := 0.0;
M[2] := 0.0;
M[3] := 0.0;
M[5] := 1.0;
M[6] := 0.0;
M[7] := 0.0;
M[9] := 0.0;
M[10] := 1.0;
M[11] := 0.0;
M[13] := 0.02686;
M[14] := 0.15515;
M[15] := 1.0;
(* '<S1>:1:56' Slist = [S1,S2,S3,S5,S6]; *)
(* MATLAB Function: '<Root>/MATLAB Function3' *)
FOR i := 0 TO 5 DO 
    Slist_tmp_0 := SINT_TO_DINT(f[i]);
    Slist[i] := DINT_TO_LREAL(Slist_tmp_0);
    Slist[i + 6] := g[i];
    Slist[i + 12] := h[i];
    Slist[i + 18] := S5[i];
    Slist[i + 24] := S6[i];
    Slist_tmp[i] := DINT_TO_SINT(Slist_tmp_0);
END_FOR;
(* '<S1>:1:62' TInverseDesired = [[1, 0, 0, X]; [0, 1, 0, Y]; [0, 0, 1, Z]; [0, 0, 0, 1]]; *)
(* MATLAB Function: '<Root>/MATLAB Function3' *)
T[0] := 1.0;
T[4] := 0.0;
T[8] := 0.0;
T[12] := r1bx;
T[1] := 0.0;
T[5] := 1.0;
T[9] := 0.0;
T[13] := r1by;
T[2] := 0.0;
T[6] := 0.0;
T[10] := 1.0;
T[14] := r1bz;
T[3] := 0.0;
T[7] := 0.0;
T[11] := 0.0;
T[15] := 1.0;
(* '<S1>:1:63' thetalist0 = [q1Inn; q2Inn; q3Inn; q5Inn; q6Inn]; *)
thetalist0[0] := q1Inn;
thetalist0[1] := q2Inn;
thetalist0[2] := q3Inn;
thetalist0[3] := q5Inn;
thetalist0[4] :=  -q1Inn;
(* '<S1>:1:64' eomg = 0.00001; *)
(* '<S1>:1:65' ev = 0.0000001; *)
(* '<S1>:1:66' [thetalist, success] = IKinSpace(Slist, M, TInverseDesired, thetalist0, eomg, ev); *)
(* *** CHAPTER 6: INVERSE KINEMATICS *** *)
(* Takes Slist: The joint screw axes in the space frame when the manipulator *)
(* is at the home position, in the format of a matrix with the *)
(* screw axes as the columns, *)
(* M: The home configuration of the end-effector, *)
(* T: The desired end-effector configuration Tsd, *)
(* thetalist0: An initial guess of joint angles that are close to  *)
(* satisfying Tsd, *)
(* eomg: A small positive tolerance on the end-effector orientation  *)
(* error. The returned joint angles must give an end-effector  *)
(* orientation error less than eomg, *)
(* ev: A small positive tolerance on the end-effector linear position  *)
(* error. The returned joint angles must give an end-effector  *)
(* position error less than ev. *)
(* Returns thetalist: Joint angles that achieve T within the specified  *)
(* tolerances, *)
(* success: A logical value where TRUE means that the function found *)
(* a solution and FALSE means that it ran through the set  *)
(* number of maximum iterations without finding a solution *)
(* within the tolerances eomg and ev. *)
(* Uses an iterative Newton-Raphson root-finding method. *)
(* The maximum number of iterations before the algorithm is terminated has  *)
(* been hardcoded in as a variable called maxiterations. It is set to 20 at  *)
(* the start of the function, but can be changed if needed.   *)
(* Example Inputs: *)
(* clear; clc; *)
(* Slist = [[0; 0;  1;  4; 0;    0], ... *)
(* [0; 0;  0;  0; 1;    0], ... *)
(* [0; 0; -1; -6; 0; -0.1]]; *)
(* M = [[-1, 0, 0, 0]; [0, 1, 0, 6]; [0, 0, -1, 2]; [0, 0, 0, 1]]; *)
(* T = [[0, 1, 0, -5]; [1, 0, 0, 4]; [0, 0, -1, 1.6858]; [0, 0, 0, 1]]; *)
(* thetalist0 = [1.5; 2.5; 3]; *)
(* eomg = 0.01; *)
(* ev = 0.001; *)
(* [thetalist, success] = IKinSpace(Slist, M, T, thetalist0, eomg, ev) *)
(* Output: *)
(* thetalist = *)
(* 1.5707 *)
(* 2.9997 *)
(* 3.1415 *)
(* success = *)
(* 1 *)
(* 'IKinSpace:48' thetalist = thetalist0; *)
(* 'IKinSpace:50' i = 0; *)
i := 0;
(* 'IKinSpace:51' maxiterations = 50; *)
(* 'IKinSpace:52' Tsb = FKinSpace(M, Slist, thetalist); *)
(* MATLAB Function: '<Root>/MATLAB Function3' *)
FOR Slist_tmp_0 := 0 TO 15 DO 
    Tsb[Slist_tmp_0] := M[Slist_tmp_0];
END_FOR;
(* *** CHAPTER 4: FORWARD KINEMATICS *** *)
(* Takes M: the home configuration (position and orientation) of the  *)
(* end-effector, *)
(* Slist: The joint screw axes in the space frame when the manipulator *)
(* is at the home position, *)
(* thetalist: A list of joint coordinates. *)
(* Returns T in SE(3) representing the end-effector frame, when the joints  *)
(* are at the specified coordinates (i.t.o Space Frame). *)
(* Example Inputs: *)
(* clear; clc; *)
(* M = [[-1, 0, 0, 0]; [0, 1, 0, 6]; [0, 0, -1, 2]; [0, 0, 0, 1]]; *)
(* Slist = [[0; 0;  1;  4; 0;    0], ... *)
(* [0; 0;  0;  0; 1;    0], ... *)
(* [0; 0; -1; -6; 0; -0.1]]; *)
(* thetalist =[pi / 2; 3; pi]; *)
(* T = FKinSpace(M, Slist, thetalist) *)
(* Output: *)
(* T = *)
(* -0.0000    1.0000         0   -5.0000 *)
(* 1.0000    0.0000         0    4.0000 *)
(* 0         0   -1.0000    1.6858 *)
(* 0         0         0    1.0000 *)
(* 'FKinSpace:27' T = M; *)
(* 'FKinSpace:28' for i = size(thetalist,1): -1: 1 *)
(* MATLAB Function: '<Root>/MATLAB Function3' *)
se3mat[0] := 0.0;
se3mat[5] := 0.0;
se3mat[10] := 0.0;
se3mat[3] := 0.0;
se3mat[7] := 0.0;
se3mat[11] := 0.0;
se3mat[15] := 0.0;
(* MATLAB Function: '<Root>/MATLAB Function3' *)
(* MATLAB Function: '<Root>/MATLAB Function3' *)
FOR c_i := 0 TO 4 DO 
    (* 'FKinSpace:29' T = MatrixExp6(VecTose3(Slist(:, i) * thetalist(i))) * T; *)
    thetalist0_0 := thetalist0[4 - c_i];
    FOR Slist_tmp_0 := 0 TO 5 DO 
        V[Slist_tmp_0] := Slist[((4 - c_i) * 6) + Slist_tmp_0] * thetalist0_0;
    END_FOR;
    (* *** CHAPTER 3: RIGID-BODY MOTIONS *** *)
    (* Takes a 6-vector (representing a spatial velocity). *)
    (* Returns the corresponding 4x4 se(3) matrix. *)
    (* Example Input: *)
    
    (* clear; clc; *)
    (* V = [1; 2; 3; 4; 5; 6]; *)
    (* se3mat = VecTose3(V) *)
    
    (* Output: *)
    (* se3mat = *)
    (* 0    -3     2     4 *)
    (* 3     0    -1     5 *)
    (* -2     1     0     6 *)
    (* 0     0     0     0  *)
    (* 'VecTose3:18' se3mat = [VecToso3(V(1: 3)), V(4: 6); 0, 0, 0, 0]; *)
    (* *** CHAPTER 3: RIGID-BODY MOTIONS *** *)
    (* Takes a 3-vector (angular velocity). *)
    (* Returns the skew symmetric matrix in so(3). *)
    (* Example Input: *)
    
    (* clear; clc; *)
    (* omg = [1; 2; 3]; *)
    (* so3mat = VecToso3(omg) *)
    
    (* Output: *)
    (* so3mat = *)
    (* 0    -3     2 *)
    (* 3     0    -1 *)
    (* -2     1     0 *)
    (* 'VecToso3:17' so3mat = [0, -omg(3), omg(2); omg(3), 0, -omg(1); -omg(2), omg(1), 0]; *)
    se3mat[4] :=  -V[2];
    se3mat[8] := V[1];
    se3mat[1] := V[2];
    se3mat[9] :=  -V[0];
    se3mat[2] :=  -V[1];
    se3mat[6] := V[0];
    se3mat[12] := V[3];
    se3mat[13] := V[4];
    se3mat[14] := V[5];
    (* *** CHAPTER 3: RIGID-BODY MOTIONS *** *)
    (* Takes a se(3) representation of exponential coordinates. *)
    (* Returns a T matrix in SE(3) that is achieved by traveling along/about the  *)
    (* screw axis S for a distance theta from an initial configuration T = I. *)
    (* Example Input: *)
    
    (* clear; clc; *)
    (* se3mat = [ 0,      0,       0,      0; *)
    (* 0,      0, -1.5708, 2.3562; *)
    (* 0, 1.5708,       0, 2.3562; *)
    (* 0,      0,       0,      0] *)
    (* T = MatrixExp6(se3mat) *)
    
    (* Output: *)
    (* T = *)
    (* 1.0000         0         0         0 *)
    (* 0    0.0000   -1.0000   -0.0000 *)
    (* 0    1.0000    0.0000    3.0000 *)
    (* 0         0         0    1.0000  *)
    (* 'MatrixExp6:22' omgtheta = so3ToVec(se3mat(1: 3, 1: 3)); *)
    (* *** CHAPTER 3: RIGID-BODY MOTIONS *** *)
    (* Takes a 3x3 skew-symmetric matrix (an element of so(3)). *)
    (* Returns the corresponding 3-vector (angular velocity). *)
    (* Example Input:  *)
    
    (* clear; clc; *)
    (* so3mat = [[0, -3, 2]; [3, 0, -1]; [-2, 1, 0]]; *)
    (* omg = so3ToVec(so3mat)   *)
    
    (* Output: *)
    (* omg = *)
    (* 1 *)
    (* 2 *)
    (* 3 *)
    (* 'so3ToVec:17' omg = [so3mat(3, 2); so3mat(1, 3); so3mat(2, 1)]; *)
    (* 'MatrixExp6:23' if NearZero(norm(omgtheta)) *)
    (* *** BASIC HELPER FUNCTIONS *** *)
    (* Takes a scalar. *)
    (* Checks if the scalar is small enough to be neglected. *)
    (* Example Input: *)
    
    (* clear; clc; *)
    (* near = -1e-7; *)
    (* judge = NearZero(near) *)
    
    (* Output: *)
    (* judge = *)
    (* 1 *)
    (* 'NearZero:15' judge = norm(near) < 1e-6; *)
    se3mat_0[0] := V[0];
    se3mat_0[1] := V[1];
    se3mat_0[2] := V[2];
    d_theta := norm(x := se3mat_0);
    IF ABS(d_theta) < 1.0E-6 THEN 
        (* 'MatrixExp6:24' T = [eye(3), se3mat(1: 3, 4); 0, 0, 0, 1]; *)
        i0_eye();
        tmp_0 := i0_eye.I;
        FOR Slist_tmp_0 := 0 TO 2 DO 
            R_tmp := DWORD_TO_DINT(SHL(DINT_TO_DWORD(Slist_tmp_0), 2));
            a[R_tmp] := tmp_0[3 * Slist_tmp_0];
            a[R_tmp + 1] := tmp_0[(3 * Slist_tmp_0) + 1];
            a[R_tmp + 2] := tmp_0[(3 * Slist_tmp_0) + 2];
            a[Slist_tmp_0 + 12] := se3mat[Slist_tmp_0 + 12];
        END_FOR;
        a[3] := 0.0;
        a[7] := 0.0;
        a[11] := 0.0;
        a[15] := 1.0;
    ELSE 
        (* 'MatrixExp6:25' else *)
        (* 'MatrixExp6:26' [omghat, theta] = AxisAng3(omgtheta); *)
        (* *** CHAPTER 3: RIGID-BODY MOTIONS *** *)
        (* Takes A 3-vector of exponential coordinates for rotation. *)
        (* Returns the unit rotation axis omghat and the corresponding rotation  *)
        (* angle theta. *)
        (* Example Input: *)
        
        (* clear; clc; *)
        (* expc3 = [1; 2; 3]; *)
        (* [omghat, theta] = AxisAng3(expc3)   *)
        
        (* Output: *)
        (* omghat = *)
        (* 0.2673 *)
        (* 0.5345 *)
        (* 0.8018 *)
        (* theta = *)
        (* 3.7417 *)
        (* 'AxisAng3:20' theta = norm(expc3); *)
        (* 'AxisAng3:21' omghat = expc3 / theta; *)
        (* 'MatrixExp6:27' omgmat = se3mat(1: 3, 1: 3) / theta; *)
        FOR Slist_tmp_0 := 0 TO 2 DO 
            omgmat_tmp := DWORD_TO_DINT(SHL(DINT_TO_DWORD(Slist_tmp_0), 2));
            omgmat[3 * Slist_tmp_0] := se3mat[omgmat_tmp] / d_theta;
            omgmat[(3 * Slist_tmp_0) + 1] := se3mat[omgmat_tmp + 1] / d_theta;
            omgmat[(3 * Slist_tmp_0) + 2] := se3mat[omgmat_tmp + 2] / d_theta;
        END_FOR;
        (* 'MatrixExp6:28' T = [MatrixExp3(se3mat(1: 3, 1: 3)), ... *)
        (* 'MatrixExp6:29'          (eye(3) * theta + (1 - cos(theta)) * omgmat ... *)
        (* 'MatrixExp6:30'           + (theta - sin(theta)) * omgmat * omgmat) ... *)
        (* 'MatrixExp6:31'             * se3mat(1: 3, 4) / theta; *)
        (* 'MatrixExp6:32'          0, 0, 0, 1]; *)
        thetalist0_0 := 1.0 - COS(d_theta);
        g_a := d_theta - SIN(d_theta);
        (* *** CHAPTER 3: RIGID-BODY MOTIONS *** *)
        (* Takes a 3x3 so(3) representation of exponential coordinates. *)
        (* Returns R in SO(3) that is achieved by rotating about omghat by theta  *)
        (* from an initial orientation R = I. *)
        (* Example Input: *)
        
        (* clear; clc; *)
        (* so3mat = [[0, -3, 2]; [3, 0, -1]; [-2, 1, 0]]; *)
        (* R = MatrixExp3(so3mat)   *)
        
        (* Output: *)
        (* R = *)
        (* -0.6949    0.7135    0.0893 *)
        (* -0.1920   -0.3038    0.9332 *)
        (* 0.6930    0.6313    0.3481 *)
        (* 'MatrixExp3:18' omgtheta = so3ToVec(so3mat); *)
        (* *** CHAPTER 3: RIGID-BODY MOTIONS *** *)
        (* Takes a 3x3 skew-symmetric matrix (an element of so(3)). *)
        (* Returns the corresponding 3-vector (angular velocity). *)
        (* Example Input:  *)
        
        (* clear; clc; *)
        (* so3mat = [[0, -3, 2]; [3, 0, -1]; [-2, 1, 0]]; *)
        (* omg = so3ToVec(so3mat)   *)
        
        (* Output: *)
        (* omg = *)
        (* 1 *)
        (* 2 *)
        (* 3 *)
        (* 'so3ToVec:17' omg = [so3mat(3, 2); so3mat(1, 3); so3mat(2, 1)]; *)
        (* 'MatrixExp3:19' if NearZero(norm(omgtheta)) *)
        (* *** BASIC HELPER FUNCTIONS *** *)
        (* Takes a scalar. *)
        (* Checks if the scalar is small enough to be neglected. *)
        (* Example Input: *)
        
        (* clear; clc; *)
        (* near = -1e-7; *)
        (* judge = NearZero(near) *)
        
        (* Output: *)
        (* judge = *)
        (* 1 *)
        (* 'NearZero:15' judge = norm(near) < 1e-6; *)
        se3mat_0[0] := V[0];
        se3mat_0[1] := V[1];
        se3mat_0[2] := V[2];
        g_theta := norm(x := se3mat_0);
        IF ABS(g_theta) < 1.0E-6 THEN 
            (* 'MatrixExp3:20' R = eye(3); *)
            i0_eye();
            b_R := i0_eye.I;
        ELSE 
            (* 'MatrixExp3:21' else *)
            (* 'MatrixExp3:22' [omghat, theta] = AxisAng3(omgtheta); *)
            (* *** CHAPTER 3: RIGID-BODY MOTIONS *** *)
            (* Takes A 3-vector of exponential coordinates for rotation. *)
            (* Returns the unit rotation axis omghat and the corresponding rotation  *)
            (* angle theta. *)
            (* Example Input: *)
            
            (* clear; clc; *)
            (* expc3 = [1; 2; 3]; *)
            (* [omghat, theta] = AxisAng3(expc3)   *)
            
            (* Output: *)
            (* omghat = *)
            (* 0.2673 *)
            (* 0.5345 *)
            (* 0.8018 *)
            (* theta = *)
            (* 3.7417 *)
            (* 'AxisAng3:20' theta = norm(expc3); *)
            (* 'AxisAng3:21' omghat = expc3 / theta; *)
            (* 'MatrixExp3:23' omgmat = so3mat / theta; *)
            FOR Slist_tmp_0 := 0 TO 2 DO 
                omgmat_tmp := DWORD_TO_DINT(SHL(DINT_TO_DWORD(Slist_tmp_0), 2));
                b_omgmat[3 * Slist_tmp_0] := se3mat[omgmat_tmp] / g_theta;
                b_omgmat[(3 * Slist_tmp_0) + 1] := se3mat[omgmat_tmp + 1] / g_theta;
                b_omgmat[(3 * Slist_tmp_0) + 2] := se3mat[omgmat_tmp + 2] / g_theta;
            END_FOR;
            (* 'MatrixExp3:24' R = eye(3) + sin(theta) * omgmat + (1 - cos(theta)) * omgmat * omgmat; *)
            l_a := SIN(g_theta);
            x_tmp := COS(g_theta);
            i0_eye();
            tmp_0 := i0_eye.I;
            FOR Slist_tmp_0 := 0 TO 2 DO 
                FOR omgmat_tmp := 0 TO 2 DO 
                    R_tmp := (3 * omgmat_tmp) + Slist_tmp_0;
                    b_R[R_tmp] := (((((1.0 - x_tmp) * b_omgmat[Slist_tmp_0 + 3]) * b_omgmat[(3 * omgmat_tmp) + 1]) + (((1.0 - x_tmp) * b_omgmat[Slist_tmp_0]) * b_omgmat[3 * omgmat_tmp])) + ((b_omgmat[Slist_tmp_0 + 6] * (1.0 - x_tmp)) * b_omgmat[(3 * omgmat_tmp) + 2])) + ((b_omgmat[R_tmp] * l_a) + tmp_0[R_tmp]);
                END_FOR;
            END_FOR;
        END_IF;
        FOR Slist_tmp_0 := 0 TO 2 DO 
            l_a := 0.0;
            FOR omgmat_tmp := 0 TO 2 DO 
                R_tmp := (3 * omgmat_tmp) + Slist_tmp_0;
                l_a := ((((((omgmat[Slist_tmp_0 + 3] * g_a) * omgmat[(3 * omgmat_tmp) + 1]) + ((g_a * omgmat[Slist_tmp_0]) * omgmat[3 * omgmat_tmp])) + ((omgmat[Slist_tmp_0 + 6] * g_a) * omgmat[(3 * omgmat_tmp) + 2])) + ((SINT_TO_LREAL(p_a[R_tmp]) * d_theta) + (omgmat[R_tmp] * thetalist0_0))) * se3mat[omgmat_tmp + 12]) + l_a;
                a[omgmat_tmp + (Slist_tmp_0 * 4)] := b_R[(3 * Slist_tmp_0) + omgmat_tmp];
            END_FOR;
            a[Slist_tmp_0 + 12] := l_a / d_theta;
        END_FOR;
        a[3] := 0.0;
        a[7] := 0.0;
        a[11] := 0.0;
        a[15] := 1.0;
    END_IF;
    FOR Slist_tmp_0 := 0 TO 3 DO 
        FOR omgmat_tmp := 0 TO 3 DO 
            a_tmp_tmp := DWORD_TO_DINT(SHL(DINT_TO_DWORD(omgmat_tmp), 2));
            R_tmp := Slist_tmp_0 + a_tmp_tmp;
            a_0[R_tmp] := 0.0;
            a_0[R_tmp] := a_0[R_tmp] + (Tsb[a_tmp_tmp] * a[Slist_tmp_0]);
            a_0[R_tmp] := (Tsb[a_tmp_tmp + 1] * a[Slist_tmp_0 + 4]) + a_0[R_tmp];
            a_0[R_tmp] := (Tsb[a_tmp_tmp + 2] * a[Slist_tmp_0 + 8]) + a_0[R_tmp];
            a_0[R_tmp] := (Tsb[a_tmp_tmp + 3] * a[Slist_tmp_0 + 12]) + a_0[R_tmp];
        END_FOR;
    END_FOR;
    FOR Slist_tmp_0 := 0 TO 15 DO 
        Tsb[Slist_tmp_0] := a_0[Slist_tmp_0];
    END_FOR;
END_FOR;
(* 'IKinSpace:53' Vs = Adjoint(Tsb) * se3ToVec(MatrixLog6(TransInv(Tsb) * T)); *)
(* *** CHAPTER 3: RIGID-BODY MOTIONS *** *)
(* Takes a transformation matrix T. *)
(* Returns its inverse.  *)
(* Uses the structure of transformation matrices to avoid taking a matrix *)
(* inverse, for efficiency. *)
(* Example Input: *)
(* clear; clc; *)
(* T = [[1, 0, 0, 0]; [0, 0, -1, 0]; [0, 1, 0, 3]; [0, 0, 0, 1]]; *)
(* invT = TransInv(T) *)
(* Ouput: *)
(* invT = *)
(* 1     0     0     0 *)
(* 0     0     1    -3 *)
(* 0    -1     0     0 *)
(* 0     0     0     1 *)
(* 'TransInv:20' [R, p] = TransToRp(T); *)
(* *** CHAPTER 3: RIGID-BODY MOTIONS *** *)
(* Takes the transformation matrix T in SE(3)  *)
(* Returns R: the corresponding rotation matrix *)
(* p: the corresponding position vector . *)
(* Example Input: *)
(* clear; clc; *)
(* T = [[1, 0, 0, 0]; [0, 0, -1, 0]; [0, 1, 0, 3]; [0, 0, 0, 1]]; *)
(* [R, p] = TransToRp(T) *)
(* Output: *)
(* R = *)
(* 1     0     0 *)
(* 0     0    -1 *)
(* 0     1     0 *)
(* p = *)
(* 0 *)
(* 0 *)
(* 3 *)
(* 'TransToRp:22' R = T(1: 3, 1: 3); *)
(* 'TransToRp:23' p = T(1: 3, 4); *)
(* 'TransInv:21' invT = [transpose(R), -transpose(R) * p; 0, 0, 0, 1]; *)
(* MATLAB Function: '<Root>/MATLAB Function3' *)
FOR Slist_tmp_0 := 0 TO 2 DO 
    omgmat[3 * Slist_tmp_0] := Tsb[Slist_tmp_0];
    omgmat[(3 * Slist_tmp_0) + 1] := Tsb[Slist_tmp_0 + 4];
    omgmat[(3 * Slist_tmp_0) + 2] := Tsb[Slist_tmp_0 + 8];
END_FOR;
(* MATLAB Function: '<Root>/MATLAB Function3' *)
FOR Slist_tmp_0 := 0 TO 8 DO 
    b_R[Slist_tmp_0] :=  -omgmat[Slist_tmp_0];
END_FOR;
(* MATLAB Function: '<Root>/MATLAB Function3' *)
FOR Slist_tmp_0 := 0 TO 2 DO 
    omgmat_tmp := DWORD_TO_DINT(SHL(DINT_TO_DWORD(Slist_tmp_0), 2));
    se3mat[omgmat_tmp] := omgmat[3 * Slist_tmp_0];
    se3mat[omgmat_tmp + 1] := omgmat[(3 * Slist_tmp_0) + 1];
    se3mat[omgmat_tmp + 2] := omgmat[(3 * Slist_tmp_0) + 2];
    se3mat[Slist_tmp_0 + 12] := (b_R[Slist_tmp_0 + 6] * Tsb[14]) + ((b_R[Slist_tmp_0 + 3] * Tsb[13]) + (b_R[Slist_tmp_0] * Tsb[12]));
END_FOR;
se3mat[3] := 0.0;
se3mat[7] := 0.0;
se3mat[11] := 0.0;
se3mat[15] := 1.0;
(* MATLAB Function: '<Root>/MATLAB Function3' *)
FOR Slist_tmp_0 := 0 TO 3 DO 
    FOR omgmat_tmp := 0 TO 3 DO 
        a_tmp_tmp := DWORD_TO_DINT(SHL(DINT_TO_DWORD(Slist_tmp_0), 2));
        R_tmp := omgmat_tmp + a_tmp_tmp;
        a_0[R_tmp] := 0.0;
        a_0[R_tmp] := a_0[R_tmp] + (T[a_tmp_tmp] * se3mat[omgmat_tmp]);
        a_0[R_tmp] := (T[a_tmp_tmp + 1] * se3mat[omgmat_tmp + 4]) + a_0[R_tmp];
        a_0[R_tmp] := (T[a_tmp_tmp + 2] * se3mat[omgmat_tmp + 8]) + a_0[R_tmp];
        a_0[R_tmp] := (T[a_tmp_tmp + 3] * se3mat[omgmat_tmp + 12]) + a_0[R_tmp];
    END_FOR;
END_FOR;
(* *** CHAPTER 3: RIGID-BODY MOTIONS *** *)
(* Takes a transformation matrix T in SE(3). *)
(* Returns the corresponding se(3) representation of exponential  *)
(* coordinates. *)
(* Example Input: *)
(* clear; clc; *)
(* T = [[1, 0, 0, 0]; [0, 0, -1, 0]; [0, 1, 0, 3]; [0, 0, 0, 1]]; *)
(* expmat = MatrixLog6(T) *)
(* Output: *)
(* expc6 = *)
(* 0         0         0         0 *)
(* 0         0   -1.5708    2.3562 *)
(* 0    1.5708         0    2.3562 *)
(* 0         0         0         0 *)
(* 'MatrixLog6:19' [R, p] = TransToRp(T); *)
(* *** CHAPTER 3: RIGID-BODY MOTIONS *** *)
(* Takes the transformation matrix T in SE(3)  *)
(* Returns R: the corresponding rotation matrix *)
(* p: the corresponding position vector . *)
(* Example Input: *)
(* clear; clc; *)
(* T = [[1, 0, 0, 0]; [0, 0, -1, 0]; [0, 1, 0, 3]; [0, 0, 0, 1]]; *)
(* [R, p] = TransToRp(T) *)
(* Output: *)
(* R = *)
(* 1     0     0 *)
(* 0     0    -1 *)
(* 0     1     0 *)
(* p = *)
(* 0 *)
(* 0 *)
(* 3 *)
(* 'TransToRp:22' R = T(1: 3, 1: 3); *)
(* 'TransToRp:23' p = T(1: 3, 4); *)
(* 'MatrixLog6:20' omgmat = MatrixLog3(R); *)
(* MATLAB Function: '<Root>/MATLAB Function3' *)
FOR Slist_tmp_0 := 0 TO 2 DO 
    R_tmp := DWORD_TO_DINT(SHL(DINT_TO_DWORD(Slist_tmp_0), 2));
    b_R[3 * Slist_tmp_0] := a_0[R_tmp];
    b_R[(3 * Slist_tmp_0) + 1] := a_0[R_tmp + 1];
    b_R[(3 * Slist_tmp_0) + 2] := a_0[R_tmp + 2];
END_FOR;
i0_MatrixLog3(b_R := b_R);
omgmat := i0_MatrixLog3.so3mat;
(* 'MatrixLog6:21' if isequal(omgmat, zeros(3)) *)
(* MATLAB Function: '<Root>/MATLAB Function3' *)
FOR Slist_tmp_0 := 0 TO 8 DO 
    tmp_0[Slist_tmp_0] := 0.0;
END_FOR;
IF isequal(varargin_1 := omgmat, varargin_2 := tmp_0) THEN 
    (* 'MatrixLog6:22' expmat = [zeros(3), T(1: 3, 4); 0, 0, 0, 0]; *)
    FOR Slist_tmp_0 := 0 TO 2 DO 
        omgmat_tmp := DWORD_TO_DINT(SHL(DINT_TO_DWORD(Slist_tmp_0), 2));
        se3mat[omgmat_tmp] := 0.0;
        se3mat[omgmat_tmp + 1] := 0.0;
        se3mat[omgmat_tmp + 2] := 0.0;
        se3mat[Slist_tmp_0 + 12] := a_0[Slist_tmp_0 + 12];
    END_FOR;
    se3mat[3] := 0.0;
    se3mat[7] := 0.0;
    se3mat[11] := 0.0;
    se3mat[15] := 0.0;
ELSE 
    (* 'MatrixLog6:23' else *)
    (* 'MatrixLog6:24' theta = acos((trace(R) - 1) / 2); *)
    theta := ACOS((((a_0[0] + a_0[5]) + a_0[10]) - 1.0) / 2.0);
    (* 'MatrixLog6:25' expmat = [omgmat, (eye(3) - omgmat / 2 ... *)
    (* 'MatrixLog6:26'                       + (1 / theta - cot(theta / 2) / 2) ... *)
    (* 'MatrixLog6:27'                         * omgmat * omgmat / theta) * p; *)
    (* 'MatrixLog6:28'               0, 0, 0, 0]; *)
    thetalist0_0 := (1.0 / theta) - ((1.0 / TAN(theta / 2.0)) / 2.0);
    i0_eye();
    tmp_0 := i0_eye.I;
    FOR Slist_tmp_0 := 0 TO 2 DO 
        se3mat_0[Slist_tmp_0] := 0.0;
        FOR omgmat_tmp := 0 TO 2 DO 
            se3mat[omgmat_tmp + (Slist_tmp_0 * 4)] := omgmat[(3 * Slist_tmp_0) + omgmat_tmp];
            R_tmp := (3 * omgmat_tmp) + Slist_tmp_0;
            se3mat_0[Slist_tmp_0] := (((((((omgmat[Slist_tmp_0 + 3] * thetalist0_0) * omgmat[(3 * omgmat_tmp) + 1]) + ((thetalist0_0 * omgmat[Slist_tmp_0]) * omgmat[3 * omgmat_tmp])) + ((omgmat[Slist_tmp_0 + 6] * thetalist0_0) * omgmat[(3 * omgmat_tmp) + 2])) / theta) + (tmp_0[R_tmp] - (omgmat[R_tmp] / 2.0))) * a_0[omgmat_tmp + 12]) + se3mat_0[Slist_tmp_0];
        END_FOR;
        se3mat[Slist_tmp_0 + 12] := se3mat_0[Slist_tmp_0];
    END_FOR;
    se3mat[3] := 0.0;
    se3mat[7] := 0.0;
    se3mat[11] := 0.0;
    se3mat[15] := 0.0;
END_IF;
(* *** CHAPTER 3: RIGID-BODY MOTIONS *** *)
(* Takes T a transformation matrix SE3.  *)
(* Returns the corresponding 6x6 adjoint representation [AdT]. *)
(* Example Input: *)
(* clear; clc; *)
(* T = [[1, 0, 0, 0]; [0, 0, -1, 0]; [0, 1, 0, 3]; [0, 0, 0, 1]]; *)
(* AdT = Adjoint(T) *)
(* Output: *)
(* AdT = *)
(* 1     0     0     0     0     0 *)
(* 0     0    -1     0     0     0 *)
(* 0     1     0     0     0     0 *)
(* 0     0     3     1     0     0 *)
(* 3     0     0     0     0    -1 *)
(* 0     0     0     0     1     0 *)
(* 'Adjoint:20' [R, p] = TransToRp(T); *)
(* *** CHAPTER 3: RIGID-BODY MOTIONS *** *)
(* Takes the transformation matrix T in SE(3)  *)
(* Returns R: the corresponding rotation matrix *)
(* p: the corresponding position vector . *)
(* Example Input: *)
(* clear; clc; *)
(* T = [[1, 0, 0, 0]; [0, 0, -1, 0]; [0, 1, 0, 3]; [0, 0, 0, 1]]; *)
(* [R, p] = TransToRp(T) *)
(* Output: *)
(* R = *)
(* 1     0     0 *)
(* 0     0    -1 *)
(* 0     1     0 *)
(* p = *)
(* 0 *)
(* 0 *)
(* 3 *)
(* 'TransToRp:22' R = T(1: 3, 1: 3); *)
(* 'TransToRp:23' p = T(1: 3, 4); *)
(* 'Adjoint:21' AdT = [R, zeros(3); VecToso3(p) * R, R]; *)
(* *** CHAPTER 3: RIGID-BODY MOTIONS *** *)
(* Takes a 3-vector (angular velocity). *)
(* Returns the skew symmetric matrix in so(3). *)
(* Example Input: *)
(* clear; clc; *)
(* omg = [1; 2; 3]; *)
(* so3mat = VecToso3(omg) *)
(* Output: *)
(* so3mat = *)
(* 0    -3     2 *)
(* 3     0    -1 *)
(* -2     1     0 *)
(* 'VecToso3:17' so3mat = [0, -omg(3), omg(2); omg(3), 0, -omg(1); -omg(2), omg(1), 0]; *)
(* *** CHAPTER 3: RIGID-BODY MOTIONS *** *)
(* Takes se3mat a 4x4 se(3) matrix *)
(* Returns the corresponding 6-vector (representing spatial velocity). *)
(* Example Input: *)
(* clear; clc; *)
(* se3mat = [[0, -3, 2, 4]; [3, 0, -1, 5]; [-2, 1, 0, 6]; [0, 0, 0, 0]]; *)
(* V = se3ToVec(se3mat) *)
(* Output: *)
(* V = *)
(* 1 *)
(* 2 *)
(* 3 *)
(* 4 *)
(* 5 *)
(* 6 *)
(* 'se3ToVec:20' V = [se3mat(3, 2); se3mat(1, 3); se3mat(2, 1); se3mat(1: 3, 4)]; *)
(* MATLAB Function: '<Root>/MATLAB Function3' *)
tmp_0[0] := 0.0;
tmp_0[3] :=  -Tsb[14];
tmp_0[6] := Tsb[13];
tmp_0[1] := Tsb[14];
tmp_0[4] := 0.0;
tmp_0[7] :=  -Tsb[12];
tmp_0[2] :=  -Tsb[13];
tmp_0[5] := Tsb[12];
tmp_0[8] := 0.0;
(* MATLAB Function: '<Root>/MATLAB Function3' *)
FOR Slist_tmp_0 := 0 TO 2 DO 
    FOR omgmat_tmp := 0 TO 2 DO 
        R_tmp := Slist_tmp_0 + (3 * omgmat_tmp);
        tmp[R_tmp] := 0.0;
        a_tmp_tmp := DWORD_TO_DINT(SHL(DINT_TO_DWORD(omgmat_tmp), 2));
        tmp[R_tmp] := tmp[R_tmp] + (Tsb[a_tmp_tmp] * tmp_0[Slist_tmp_0]);
        tmp[R_tmp] := (Tsb[a_tmp_tmp + 1] * tmp_0[Slist_tmp_0 + 3]) + tmp[R_tmp];
        tmp[R_tmp] := (Tsb[a_tmp_tmp + 2] * tmp_0[Slist_tmp_0 + 6]) + tmp[R_tmp];
        Tsb_0[omgmat_tmp + (6 * Slist_tmp_0)] := Tsb[(Slist_tmp_0 * 4) + omgmat_tmp];
        Tsb_0[omgmat_tmp + (6 * (Slist_tmp_0 + 3))] := 0.0;
    END_FOR;
END_FOR;
(* MATLAB Function: '<Root>/MATLAB Function3' *)
V[0] := se3mat[6];
V[1] := se3mat[8];
V[2] := se3mat[1];
FOR Slist_tmp_0 := 0 TO 2 DO 
    Tsb_0[(6 * Slist_tmp_0) + 3] := tmp[3 * Slist_tmp_0];
    omgmat_tmp := DWORD_TO_DINT(SHL(DINT_TO_DWORD(Slist_tmp_0), 2));
    R_tmp := 6 * (Slist_tmp_0 + 3);
    Tsb_0[R_tmp + 3] := Tsb[omgmat_tmp];
    Tsb_0[(6 * Slist_tmp_0) + 4] := tmp[(3 * Slist_tmp_0) + 1];
    Tsb_0[R_tmp + 4] := Tsb[omgmat_tmp + 1];
    Tsb_0[(6 * Slist_tmp_0) + 5] := tmp[(3 * Slist_tmp_0) + 2];
    Tsb_0[R_tmp + 5] := Tsb[omgmat_tmp + 2];
    V[Slist_tmp_0 + 3] := se3mat[Slist_tmp_0 + 12];
END_FOR;
(* MATLAB Function: '<Root>/MATLAB Function3' *)
FOR Slist_tmp_0 := 0 TO 5 DO 
    Vs[Slist_tmp_0] := 0.0;
    FOR omgmat_tmp := 0 TO 5 DO 
        Vs[Slist_tmp_0] := (Tsb_0[(6 * omgmat_tmp) + Slist_tmp_0] * V[omgmat_tmp]) + Vs[Slist_tmp_0];
    END_FOR;
END_FOR;
(* 'IKinSpace:54' err = norm(Vs(1: 3)) > eomg || norm(Vs(4: 6)) > ev; *)
(* MATLAB Function: '<Root>/MATLAB Function3' *)
se3mat_0[0] := Vs[0];
se3mat_0[1] := Vs[1];
se3mat_0[2] := Vs[2];
IF norm(x := se3mat_0) > 1.0E-5 THEN 
    err := TRUE;
ELSE 
    se3mat_0[0] := Vs[3];
    se3mat_0[1] := Vs[4];
    se3mat_0[2] := Vs[5];
    IF norm(x := se3mat_0) > 1.0E-7 THEN 
        err := TRUE;
    ELSE 
        err := FALSE;
    END_IF;
END_IF;
(* 'IKinSpace:55' while err && i < maxiterations *)
IF err THEN 
    tmp_3[0] := 0.0;
    tmp_3[4] := 0.0;
    tmp_3[8] := 0.0;
    tmp_5[0] := 0.0;
    tmp_5[4] := 0.0;
    tmp_5[8] := 0.0;
    FOR Slist_tmp_0 := 0 TO 8 DO 
        tmp_4[Slist_tmp_0] := 0.0;
    END_FOR;
END_IF;
WHILE err AND (i < 50) DO
    (* 'IKinSpace:56' thetalist = thetalist + pinv(JacobianSpace(Slist, thetalist)) * Vs; *)
    (* *** CHAPTER 5: VELOCITY KINEMATICS AND STATICS *** *)
    (* Takes Slist: The joint screw axes in the space frame when the manipulator *)
    (* is at the home position, in the format of a matrix with the *)
    (* screw axes as the columns, *)
    (* thetalist: A list of joint coordinates.  *)
    (* Returns the corresponding space Jacobian (6xn real numbers). *)
    (* Example Input: *)
    
    (* clear; clc; *)
    (* Slist = [[0; 0; 1;   0; 0.2; 0.2], ... *)
    (* [1; 0; 0;   2;   0;   3], ... *)
    (* [0; 1; 0;   0;   2;   1], ... *)
    (* [1; 0; 0; 0.2; 0.3; 0.4]]; *)
    (* thetalist = [0.2; 1.1; 0.1; 1.2]; *)
    (* Js = JacobianSpace(Slist, thetalist) *)
    
    (* Output: *)
    (* Js = *)
    (* 0    0.9801   -0.0901    0.9575 *)
    (* 0    0.1987    0.4446    0.2849 *)
    (* 1.0000         0    0.8912   -0.0453 *)
    (* 0    1.9522   -2.2164   -0.5116 *)
    (* 0.2000    0.4365   -2.4371    2.7754 *)
    (* 0.2000    2.9603    3.2357    2.2251 *)
    (* 'JacobianSpace:27' Js = Slist; *)
    FOR Slist_tmp_0 := 0 TO 29 DO 
        Js[Slist_tmp_0] := Slist[Slist_tmp_0];
    END_FOR;
    (* 'JacobianSpace:28' T = eye(4); *)
    FOR Slist_tmp_0 := 0 TO 15 DO 
        a_0[Slist_tmp_0] := 0.0;
    END_FOR;
    a_0[0] := 1.0;
    a_0[5] := 1.0;
    a_0[10] := 1.0;
    a_0[15] := 1.0;
    (* 'JacobianSpace:29' for i = 2: length(thetalist) *)
    se3mat[0] := 0.0;
    se3mat[5] := 0.0;
    se3mat[10] := 0.0;
    se3mat[3] := 0.0;
    se3mat[7] := 0.0;
    se3mat[11] := 0.0;
    se3mat[15] := 0.0;
    FOR d_i := 0 TO 3 DO 
        (* 'JacobianSpace:30' T = T * MatrixExp6(VecTose3(Slist(:, i - 1) * thetalist(i - 1))); *)
        thetalist0_0 := thetalist0[d_i];
        FOR Slist_tmp_0 := 0 TO 5 DO 
            V[Slist_tmp_0] := Slist[(6 * d_i) + Slist_tmp_0] * thetalist0_0;
        END_FOR;
        (* *** CHAPTER 3: RIGID-BODY MOTIONS *** *)
        (* Takes a 6-vector (representing a spatial velocity). *)
        (* Returns the corresponding 4x4 se(3) matrix. *)
        (* Example Input: *)
        
        (* clear; clc; *)
        (* V = [1; 2; 3; 4; 5; 6]; *)
        (* se3mat = VecTose3(V) *)
        
        (* Output: *)
        (* se3mat = *)
        (* 0    -3     2     4 *)
        (* 3     0    -1     5 *)
        (* -2     1     0     6 *)
        (* 0     0     0     0  *)
        (* 'VecTose3:18' se3mat = [VecToso3(V(1: 3)), V(4: 6); 0, 0, 0, 0]; *)
        (* *** CHAPTER 3: RIGID-BODY MOTIONS *** *)
        (* Takes a 3-vector (angular velocity). *)
        (* Returns the skew symmetric matrix in so(3). *)
        (* Example Input: *)
        
        (* clear; clc; *)
        (* omg = [1; 2; 3]; *)
        (* so3mat = VecToso3(omg) *)
        
        (* Output: *)
        (* so3mat = *)
        (* 0    -3     2 *)
        (* 3     0    -1 *)
        (* -2     1     0 *)
        (* 'VecToso3:17' so3mat = [0, -omg(3), omg(2); omg(3), 0, -omg(1); -omg(2), omg(1), 0]; *)
        se3mat[4] :=  -V[2];
        se3mat[8] := V[1];
        se3mat[1] := V[2];
        se3mat[9] :=  -V[0];
        se3mat[2] :=  -V[1];
        se3mat[6] := V[0];
        se3mat[12] := V[3];
        se3mat[13] := V[4];
        se3mat[14] := V[5];
        (* *** CHAPTER 3: RIGID-BODY MOTIONS *** *)
        (* Takes a se(3) representation of exponential coordinates. *)
        (* Returns a T matrix in SE(3) that is achieved by traveling along/about the  *)
        (* screw axis S for a distance theta from an initial configuration T = I. *)
        (* Example Input: *)
        
        (* clear; clc; *)
        (* se3mat = [ 0,      0,       0,      0; *)
        (* 0,      0, -1.5708, 2.3562; *)
        (* 0, 1.5708,       0, 2.3562; *)
        (* 0,      0,       0,      0] *)
        (* T = MatrixExp6(se3mat) *)
        
        (* Output: *)
        (* T = *)
        (* 1.0000         0         0         0 *)
        (* 0    0.0000   -1.0000   -0.0000 *)
        (* 0    1.0000    0.0000    3.0000 *)
        (* 0         0         0    1.0000  *)
        (* 'MatrixExp6:22' omgtheta = so3ToVec(se3mat(1: 3, 1: 3)); *)
        (* *** CHAPTER 3: RIGID-BODY MOTIONS *** *)
        (* Takes a 3x3 skew-symmetric matrix (an element of so(3)). *)
        (* Returns the corresponding 3-vector (angular velocity). *)
        (* Example Input:  *)
        
        (* clear; clc; *)
        (* so3mat = [[0, -3, 2]; [3, 0, -1]; [-2, 1, 0]]; *)
        (* omg = so3ToVec(so3mat)   *)
        
        (* Output: *)
        (* omg = *)
        (* 1 *)
        (* 2 *)
        (* 3 *)
        (* 'so3ToVec:17' omg = [so3mat(3, 2); so3mat(1, 3); so3mat(2, 1)]; *)
        (* 'MatrixExp6:23' if NearZero(norm(omgtheta)) *)
        (* *** BASIC HELPER FUNCTIONS *** *)
        (* Takes a scalar. *)
        (* Checks if the scalar is small enough to be neglected. *)
        (* Example Input: *)
        
        (* clear; clc; *)
        (* near = -1e-7; *)
        (* judge = NearZero(near) *)
        
